   1:L PR[91] 10mm/sec CNT100;
   1:  PR[GP1:91,1] = PR[GP1:90,1] + 67.778;
   1:  PR[GP1:91,2] = PR[GP1:90,2] + -19.376;
   1:L PR[91] 10mm/sec CNT100;
   1:  PR[GP1:91,1] = PR[GP1:90,1] + 70.791;
   1:  PR[GP1:91,2] = PR[GP1:90,2] + -14.501;
   1:L PR[91] 10mm/sec CNT100;
   1:  PR[GP1:91,1] = PR[GP1:90,1] + 71.584;
   1:  PR[GP1:91,2] = PR[GP1:90,2] + -10.994;
   1:L PR[91] 10mm/sec CNT100;
   1:  PR[GP1:91,1] = PR[GP1:90,1] + 73.496;
   1:  PR[GP1:91,2] = PR[GP1:90,2] + -5.450;
   1:L PR[91] 10mm/sec CNT100;
   1:  PR[GP1:91,1] = PR[GP1:90,1] + 74.129;
   1:  PR[GP1:91,2] = PR[GP1:90,2] + 0.245;
   1:L PR[91] 10mm/sec CNT100;
   1:  PR[GP1:91,1] = PR[GP1:90,1] + 73.337;
   1:  PR[GP1:91,2] = PR[GP1:90,2] + 3.752;
   1:L PR[91] 10mm/sec CNT100;
   1:  PR[GP1:91,1] = PR[GP1:90,1] + 72.689;
   1:  PR[GP1:91,2] = PR[GP1:90,2] + 9.581;
   1:L PR[91] 10mm/sec CNT100;
   1:  PR[GP1:91,1] = PR[GP1:90,1] + 70.809;
   1:  PR[GP1:91,2] = PR[GP1:90,2] + 15.031;
   1:L PR[91] 10mm/sec CNT100;
   1:  PR[GP1:91,1] = PR[GP1:90,1] + 67.761;
   1:  PR[GP1:91,2] = PR[GP1:90,2] + 19.962;
   1:L PR[91] 10mm/sec CNT100;
   1:  PR[GP1:91,1] = PR[GP1:90,1] + 65.538;
   1:  PR[GP1:91,2] = PR[GP1:90,2] + 22.788;
   1:L PR[91] 10mm/sec CNT100;
   1:  PR[GP1:91,1] = PR[GP1:90,1] + 61.480;
   1:  PR[GP1:91,2] = PR[GP1:90,2] + 26.931;
   1:L PR[91] 10mm/sec CNT100;
   1:  PR[GP1:91,1] = PR[GP1:90,1] + 56.613;
   1:  PR[GP1:91,2] = PR[GP1:90,2] + 30.080;
   1:L PR[91] 10mm/sec CNT100;
   1:  PR[GP1:91,1] = PR[GP1:90,1] + 53.392;
   1:  PR[GP1:91,2] = PR[GP1:90,2] + 31.677;
   1:L PR[91] 10mm/sec CNT100;
   1:  PR[GP1:91,1] = PR[GP1:90,1] + 47.950;
   1:  PR[GP1:91,2] = PR[GP1:90,2] + 33.680;
   1:L PR[91] 10mm/sec CNT100;
   1:  PR[GP1:91,1] = PR[GP1:90,1] + 42.203;
   1:  PR[GP1:91,2] = PR[GP1:90,2] + 34.439;
   1:L PR[91] 10mm/sec CNT100;
   1:  PR[GP1:91,1] = PR[GP1:90,1] + 38.606;
   1:  PR[GP1:91,2] = PR[GP1:90,2] + 34.497;
   1:L PR[91] 10mm/sec CNT100;
   1:  PR[GP1:91,1] = PR[GP1:90,1] + 32.831;
   1:  PR[GP1:91,2] = PR[GP1:90,2] + 33.975;
   1:L PR[91] 10mm/sec CNT100;
   1:  PR[GP1:91,1] = PR[GP1:90,1] + 27.313;
   1:  PR[GP1:91,2] = PR[GP1:90,2] + 32.198;
   1:L PR[91] 10mm/sec CNT100;
   1:  PR[GP1:91,1] = PR[GP1:90,1] + 24.043;
   1:  PR[GP1:91,2] = PR[GP1:90,2] + 30.704;
   1:L PR[91] 10mm/sec CNT100;
   1:  PR[GP1:91,1] = PR[GP1:90,1] + 19.047;
   1:  PR[GP1:91,2] = PR[GP1:90,2] + 27.757;
   1:L PR[91] 10mm/sec CNT100;
   1:  PR[GP1:91,1] = PR[GP1:90,1] + 14.824;
   1:  PR[GP1:91,2] = PR[GP1:90,2] + 23.787;
   1:L PR[91] 10mm/sec CNT100;
   1:  PR[GP1:91,1] = PR[GP1:90,1] + 12.513;
   1:  PR[GP1:91,2] = PR[GP1:90,2] + 21.033;
   1:L PR[91] 10mm/sec CNT100;
   1:  PR[GP1:91,1] = PR[GP1:90,1] + 9.263;
   1:  PR[GP1:91,2] = PR[GP1:90,2] + 16.229;
   1:L PR[91] 10mm/sec CNT100;
   1:  PR[GP1:91,1] = PR[GP1:90,1] + 7.149;
   1:  PR[GP1:91,2] = PR[GP1:90,2] + 10.833;
   1:L PR[91] 10mm/sec CNT100;
   1:  PR[GP1:91,1] = PR[GP1:90,1] + 6.245;
   1:  PR[GP1:91,2] = PR[GP1:90,2] + 7.355;
   1:L PR[91] 10mm/sec CNT100;
   1:  PR[GP1:91,1] = PR[GP1:90,1] + 5.362;
   1:  PR[GP1:91,2] = PR[GP1:90,2] + 1.589;
   1:L PR[91] 10mm/sec CNT100;
   1:  PR[GP1:91,1] = PR[GP1:90,1] + 5.334;
   1:  PR[GP1:91,2] = PR[GP1:90,2] + 0.841;
   1:L PR[91] 10mm/sec CNT100;
   1:  PR[GP1:91,1] = PR[GP1:90,1] + -5.749;
   1:  PR[GP1:91,2] = PR[GP1:90,2] + 0.842;
   1:L PR[91] 10mm/sec CNT100;
   1:  PR[GP1:91,1] = PR[GP1:90,1] + -6.245;
   1:  PR[GP1:91,2] = PR[GP1:90,2] + 2.791;
   1:L PR[91] 10mm/sec CNT100;
   1:  PR[GP1:91,1] = PR[GP1:90,1] + -6.800;
   1:  PR[GP1:91,2] = PR[GP1:90,2] + 5.072;
   1:L PR[91] 10mm/sec CNT100;
   1:  PR[GP1:91,1] = PR[GP1:90,1] + -7.686;
   1:  PR[GP1:91,2] = PR[GP1:90,2] + 10.862;
   1:L PR[91] 10mm/sec CNT100;
   1:  PR[GP1:91,1] = PR[GP1:90,1] + -9.778;
   1:  PR[GP1:91,2] = PR[GP1:90,2] + 16.200;
   1:L PR[91] 10mm/sec CNT100;
   1:  PR[GP1:91,1] = PR[GP1:90,1] + -12.088;
   1:  PR[GP1:91,2] = PR[GP1:90,2] + 18.953;
   1:L PR[91] 10mm/sec CNT100;
   1:  PR[GP1:91,1] = PR[GP1:90,1] + -15.374;
   1:  PR[GP1:91,2] = PR[GP1:90,2] + 23.809;
   1:L PR[91] 10mm/sec CNT100;
   1:  PR[GP1:91,1] = PR[GP1:90,1] + -19.550;
   1:  PR[GP1:91,2] = PR[GP1:90,2] + 27.735;
   1:L PR[91] 10mm/sec CNT100;
   1:  PR[GP1:91,1] = PR[GP1:90,1] + -22.820;
   1:  PR[GP1:91,2] = PR[GP1:90,2] + 29.228;
   1:L PR[91] 10mm/sec CNT100;
   1:  PR[GP1:91,1] = PR[GP1:90,1] + -27.870;
   1:  PR[GP1:91,2] = PR[GP1:90,2] + 32.208;
   1:L PR[91] 10mm/sec CNT100;
   1:  PR[GP1:91,1] = PR[GP1:90,1] + -33.326;
   1:  PR[GP1:91,2] = PR[GP1:90,2] + 33.965;
   1:L PR[91] 10mm/sec CNT100;
   1:  PR[GP1:91,1] = PR[GP1:90,1] + -36.922;
   1:  PR[GP1:91,2] = PR[GP1:90,2] + 33.908;
   1:L PR[91] 10mm/sec CNT100;
   1:  PR[GP1:91,1] = PR[GP1:90,1] + -42.761;
   1:  PR[GP1:91,2] = PR[GP1:90,2] + 34.435;
   1:L PR[91] 10mm/sec CNT100;
   1:  PR[GP1:91,1] = PR[GP1:90,1] + -48.444;
   1:  PR[GP1:91,2] = PR[GP1:90,2] + 33.685;
   1:L PR[91] 10mm/sec CNT100;
   1:  PR[GP1:91,1] = PR[GP1:90,1] + -51.664;
   1:  PR[GP1:91,2] = PR[GP1:90,2] + 32.088;
   1:L PR[91] 10mm/sec CNT100;
   1:  PR[GP1:91,1] = PR[GP1:90,1] + -57.167;
   1:  PR[GP1:91,2] = PR[GP1:90,2] + 30.062;
   1:L PR[91] 10mm/sec CNT100;
   1:  PR[GP1:91,1] = PR[GP1:90,1] + -61.979;
   1:  PR[GP1:91,2] = PR[GP1:90,2] + 26.949;
   1:L PR[91] 10mm/sec CNT100;
   1:  PR[GP1:91,1] = PR[GP1:90,1] + -64.201;
   1:  PR[GP1:91,2] = PR[GP1:90,2] + 24.123;
   1:L PR[91] 10mm/sec CNT100;
   1:  PR[GP1:91,1] = PR[GP1:90,1] + -68.304;
   1:  PR[GP1:91,2] = PR[GP1:90,2] + 19.934;
   1:L PR[91] 10mm/sec CNT100;
   1:  PR[GP1:91,1] = PR[GP1:90,1] + -71.318;
   1:  PR[GP1:91,2] = PR[GP1:90,2] + 15.059;
   1:L PR[91] 10mm/sec CNT100;
   1:  PR[GP1:91,1] = PR[GP1:90,1] + -72.110;
   1:  PR[GP1:91,2] = PR[GP1:90,2] + 11.552;
   1:L PR[91] 10mm/sec CNT100;
   1:  PR[GP1:91,1] = PR[GP1:90,1] + -74.022;
   1:  PR[GP1:91,2] = PR[GP1:90,2] + 6.008;
   1:L PR[91] 10mm/sec CNT100;
   1:  PR[GP1:91,1] = PR[GP1:90,1] + -74.656;
   1:  PR[GP1:91,2] = PR[GP1:90,2] + 0.313;
   1:L PR[91] 10mm/sec CNT100;
   1:  PR[GP1:91,1] = PR[GP1:90,1] + -73.863;
   1:  PR[GP1:91,2] = PR[GP1:90,2] + -3.194;
   1:L PR[91] 10mm/sec CNT100;
   1:  PR[GP1:91,1] = PR[GP1:90,1] + -73.215;
   1:  PR[GP1:91,2] = PR[GP1:90,2] + -9.023;
   1:L PR[91] 10mm/sec CNT100;
   1:  PR[GP1:91,1] = PR[GP1:90,1] + -71.335;
   1:  PR[GP1:91,2] = PR[GP1:90,2] + -14.473;
   1:L PR[91] 10mm/sec CNT100;
   1:  PR[GP1:91,1] = PR[GP1:90,1] + -68.287;
   1:  PR[GP1:91,2] = PR[GP1:90,2] + -19.404;
   1:L PR[91] 10mm/sec CNT100;
   1:  PR[GP1:91,1] = PR[GP1:90,1] + -66.065;
   1:  PR[GP1:91,2] = PR[GP1:90,2] + -22.230;
   1:L PR[91] 10mm/sec CNT100;
   1:  PR[GP1:91,1] = PR[GP1:90,1] + -62.007;
   1:  PR[GP1:91,2] = PR[GP1:90,2] + -26.373;
   1:L PR[91] 10mm/sec CNT100;
   1:  PR[GP1:91,1] = PR[GP1:90,1] + -57.140;
   1:  PR[GP1:91,2] = PR[GP1:90,2] + -29.522;
   1:L PR[91] 10mm/sec CNT100;
   1:  PR[GP1:91,1] = PR[GP1:90,1] + -53.918;
   1:  PR[GP1:91,2] = PR[GP1:90,2] + -31.119;
   1:L PR[91] 10mm/sec CNT100;
   1:  PR[GP1:91,1] = PR[GP1:90,1] + -48.476;
   1:  PR[GP1:91,2] = PR[GP1:90,2] + -33.122;
   1:L PR[91] 10mm/sec CNT100;
   1:  PR[GP1:91,1] = PR[GP1:90,1] + -42.729;
   1:  PR[GP1:91,2] = PR[GP1:90,2] + -33.881;
   1:L PR[91] 10mm/sec CNT100;
   1:  PR[GP1:91,1] = PR[GP1:90,1] + -39.133;
   1:  PR[GP1:91,2] = PR[GP1:90,2] + -33.939;
   1:L PR[91] 10mm/sec CNT100;
   1:  PR[GP1:91,1] = PR[GP1:90,1] + -33.357;
   1:  PR[GP1:91,2] = PR[GP1:90,2] + -33.417;
   1:L PR[91] 10mm/sec CNT100;
   1:  PR[GP1:91,1] = PR[GP1:90,1] + -27.840;
   1:  PR[GP1:91,2] = PR[GP1:90,2] + -31.640;
   1:L PR[91] 10mm/sec CNT100;
   1:  PR[GP1:91,1] = PR[GP1:90,1] + -24.569;
   1:  PR[GP1:91,2] = PR[GP1:90,2] + -30.146;
   1:L PR[91] 10mm/sec CNT100;
   1:  PR[GP1:91,1] = PR[GP1:90,1] + -19.574;
   1:  PR[GP1:91,2] = PR[GP1:90,2] + -27.199;
   1:L PR[91] 10mm/sec CNT100;
   1:  PR[GP1:91,1] = PR[GP1:90,1] + -15.351;
   1:  PR[GP1:91,2] = PR[GP1:90,2] + -23.229;
   1:L PR[91] 10mm/sec CNT100;
   1:  PR[GP1:91,1] = PR[GP1:90,1] + -13.039;
   1:  PR[GP1:91,2] = PR[GP1:90,2] + -20.475;
   1:L PR[91] 10mm/sec CNT100;
   1:  PR[GP1:91,1] = PR[GP1:90,1] + -9.789;
   1:  PR[GP1:91,2] = PR[GP1:90,2] + -15.671;
   1:L PR[91] 10mm/sec CNT100;
   1:  PR[GP1:91,1] = PR[GP1:90,1] + -7.675;
   1:  PR[GP1:91,2] = PR[GP1:90,2] + -10.275;
   1:L PR[91] 10mm/sec CNT100;
   1:  PR[GP1:91,1] = PR[GP1:90,1] + -6.771;
   1:  PR[GP1:91,2] = PR[GP1:90,2] + -6.797;
   1:L PR[91] 10mm/sec CNT100;
   1:  PR[GP1:91,1] = PR[GP1:90,1] + -5.888;
   1:  PR[GP1:91,2] = PR[GP1:90,2] + -1.031;
   1:L PR[91] 10mm/sec CNT100;
   1:  PR[GP1:91,1] = PR[GP1:90,1] + -5.861;
   1:  PR[GP1:91,2] = PR[GP1:90,2] + -0.283;
   1:L PR[91] 10mm/sec CNT100;
   1:  PR[GP1:91,1] = PR[GP1:90,1] + 5.223;
   1:  PR[GP1:91,2] = PR[GP1:90,2] + -0.284;
   1:L PR[91] 10mm/sec CNT100;
   1:  PR[GP1:91,1] = PR[GP1:90,1] + 5.979;
   1:  PR[GP1:91,2] = PR[GP1:90,2] + -3.401;
   1:  PR[GP1:91,3] = PR[GP1:90,3] + 7.015;
   1:L PR[91] 10mm/sec CNT100;
   1:  PR[GP1:91,1] = PR[GP1:90,1] + 6.955;
   1:  PR[GP1:91,2] = PR[GP1:90,2] + -9.774;
   1:L PR[91] 10mm/sec CNT100;
   1:  PR[GP1:91,1] = PR[GP1:90,1] + 9.261;
   1:  PR[GP1:91,2] = PR[GP1:90,2] + -15.661;
   1:L PR[91] 10mm/sec CNT100;
   1:  PR[GP1:91,1] = PR[GP1:90,1] + 10.816;
   1:  PR[GP1:91,2] = PR[GP1:90,2] + -17.514;
   1:L PR[91] 10mm/sec CNT100;
   1:  PR[GP1:91,1] = PR[GP1:90,1] + 14.432;
   1:  PR[GP1:91,2] = PR[GP1:90,2] + -22.857;
   1:L PR[91] 10mm/sec CNT100;
   1:  PR[GP1:91,1] = PR[GP1:90,1] + 19.038;
   1:  PR[GP1:91,2] = PR[GP1:90,2] + -27.188;
   1:L PR[91] 10mm/sec CNT100;
   1:  PR[GP1:91,1] = PR[GP1:90,1] + 21.239;
   1:  PR[GP1:91,2] = PR[GP1:90,2] + -28.193;
   1:L PR[91] 10mm/sec CNT100;
   1:  PR[GP1:91,1] = PR[GP1:90,1] + 26.796;
   1:  PR[GP1:91,2] = PR[GP1:90,2] + -31.472;
   1:L PR[91] 10mm/sec CNT100;
   1:  PR[GP1:91,1] = PR[GP1:90,1] + 32.814;
   1:  PR[GP1:91,2] = PR[GP1:90,2] + -33.410;
   1:L PR[91] 10mm/sec CNT100;
   1:  PR[GP1:91,1] = PR[GP1:90,1] + 35.234;
   1:  PR[GP1:91,2] = PR[GP1:90,2] + -33.371;
   1:L PR[91] 10mm/sec CNT100;
   1:  PR[GP1:91,1] = PR[GP1:90,1] + 41.660;
   1:  PR[GP1:91,2] = PR[GP1:90,2] + -33.952;
   1:L PR[91] 10mm/sec CNT100;
   1:  PR[GP1:91,1] = PR[GP1:90,1] + 47.927;
   1:  PR[GP1:91,2] = PR[GP1:90,2] + -33.124;
   1:L PR[91] 10mm/sec CNT100;
   1:  PR[GP1:91,1] = PR[GP1:90,1] + 50.095;
   1:  PR[GP1:91,2] = PR[GP1:90,2] + -32.050;
   1:L PR[91] 10mm/sec CNT100;
   1:  PR[GP1:91,1] = PR[GP1:90,1] + 56.151;
   1:  PR[GP1:91,2] = PR[GP1:90,2] + -29.820;
   1:L PR[91] 10mm/sec CNT100;
   1:  PR[GP1:91,1] = PR[GP1:90,1] + 61.458;
   1:  PR[GP1:91,2] = PR[GP1:90,2] + -26.386;
   1:L PR[91] 10mm/sec CNT100;
   1:  PR[GP1:91,1] = PR[GP1:90,1] + 62.953;
   1:  PR[GP1:91,2] = PR[GP1:90,2] + -24.485;
   1:L PR[91] 10mm/sec CNT100;
   1:  PR[GP1:91,1] = PR[GP1:90,1] + 67.470;
   1:  PR[GP1:91,2] = PR[GP1:90,2] + -19.875;
   1:L PR[91] 10mm/sec CNT100;
   1:  PR[GP1:91,1] = PR[GP1:90,1] + 70.793;
   1:  PR[GP1:91,2] = PR[GP1:90,2] + -14.498;
   1:L PR[91] 10mm/sec CNT100;
   1:  PR[GP1:91,1] = PR[GP1:90,1] + 71.326;
   1:  PR[GP1:91,2] = PR[GP1:90,2] + -12.138;
   1:L PR[91] 10mm/sec CNT100;
   1:  PR[GP1:91,1] = PR[GP1:90,1] + 73.431;
   1:  PR[GP1:91,2] = PR[GP1:90,2] + -6.036;
   1:L PR[91] 10mm/sec CNT100;
   1:  PR[GP1:91,1] = PR[GP1:90,1] + 74.129;
   1:  PR[GP1:91,2] = PR[GP1:90,2] + 0.245;
   1:L PR[91] 10mm/sec CNT100;
   1:  PR[GP1:91,1] = PR[GP1:90,1] + 73.596;
   1:  PR[GP1:91,2] = PR[GP1:90,2] + 2.605;
   1:L PR[91] 10mm/sec CNT100;
   1:  PR[GP1:91,1] = PR[GP1:90,1] + 72.883;
   1:  PR[GP1:91,2] = PR[GP1:90,2] + 9.020;
   1:L PR[91] 10mm/sec CNT100;
   1:  PR[GP1:91,1] = PR[GP1:90,1] + 70.811;
   1:  PR[GP1:91,2] = PR[GP1:90,2] + 15.027;
   1:L PR[91] 10mm/sec CNT100;
   1:  PR[GP1:91,1] = PR[GP1:90,1] + 67.452;
   1:  PR[GP1:91,2] = PR[GP1:90,2] + 20.461;
   1:L PR[91] 10mm/sec CNT100;
   1:  PR[GP1:91,1] = PR[GP1:90,1] + 65.957;
   1:  PR[GP1:91,2] = PR[GP1:90,2] + 22.363;
   1:L PR[91] 10mm/sec CNT100;
   1:  PR[GP1:91,1] = PR[GP1:90,1] + 61.486;
   1:  PR[GP1:91,2] = PR[GP1:90,2] + 26.926;
   1:L PR[91] 10mm/sec CNT100;
   1:  PR[GP1:91,1] = PR[GP1:90,1] + 56.124;
   1:  PR[GP1:91,2] = PR[GP1:90,2] + 30.395;
   1:L PR[91] 10mm/sec CNT100;
   1:  PR[GP1:91,1] = PR[GP1:90,1] + 53.955;
   1:  PR[GP1:91,2] = PR[GP1:90,2] + 31.470;
   1:L PR[91] 10mm/sec CNT100;
   1:  PR[GP1:91,1] = PR[GP1:90,1] + 47.960;
   1:  PR[GP1:91,2] = PR[GP1:90,2] + 33.678;
   1:L PR[91] 10mm/sec CNT100;
   1:  PR[GP1:91,1] = PR[GP1:90,1] + 41.629;
   1:  PR[GP1:91,2] = PR[GP1:90,2] + 34.514;
   1:L PR[91] 10mm/sec CNT100;
   1:  PR[GP1:91,1] = PR[GP1:90,1] + 39.208;
   1:  PR[GP1:91,2] = PR[GP1:90,2] + 34.553;
   1:L PR[91] 10mm/sec CNT100;
   1:  PR[GP1:91,1] = PR[GP1:90,1] + 32.845;
   1:  PR[GP1:91,2] = PR[GP1:90,2] + 33.978;
   1:L PR[91] 10mm/sec CNT100;
   1:  PR[GP1:91,1] = PR[GP1:90,1] + 26.766;
   1:  PR[GP1:91,2] = PR[GP1:90,2] + 32.020;
   1:L PR[91] 10mm/sec CNT100;
   1:  PR[GP1:91,1] = PR[GP1:90,1] + 24.565;
   1:  PR[GP1:91,2] = PR[GP1:90,2] + 31.015;
   1:L PR[91] 10mm/sec CNT100;
   1:  PR[GP1:91,1] = PR[GP1:90,1] + 19.062;
   1:  PR[GP1:91,2] = PR[GP1:90,2] + 27.768;
   1:L PR[91] 10mm/sec CNT100;
   1:  PR[GP1:91,1] = PR[GP1:90,1] + 14.409;
   1:  PR[GP1:91,2] = PR[GP1:90,2] + 23.394;
   1:L PR[91] 10mm/sec CNT100;
   1:  PR[GP1:91,1] = PR[GP1:90,1] + 12.853;
   1:  PR[GP1:91,2] = PR[GP1:90,2] + 21.541;
   1:L PR[91] 10mm/sec CNT100;
   1:  PR[GP1:91,1] = PR[GP1:90,1] + 9.273;
   1:  PR[GP1:91,2] = PR[GP1:90,2] + 16.248;
   1:L PR[91] 10mm/sec CNT100;
   1:  PR[GP1:91,1] = PR[GP1:90,1] + 6.943;
   1:  PR[GP1:91,2] = PR[GP1:90,2] + 10.303;
   1:L PR[91] 10mm/sec CNT100;
   1:  PR[GP1:91,1] = PR[GP1:90,1] + 6.335;
   1:  PR[GP1:91,2] = PR[GP1:90,2] + 7.962;
   1:L PR[91] 10mm/sec CNT100;
   1:  PR[GP1:91,1] = PR[GP1:90,1] + 5.363;
   1:  PR[GP1:91,2] = PR[GP1:90,2] + 1.613;
   1:L PR[91] 10mm/sec CNT100;
   1:  PR[GP1:91,1] = PR[GP1:90,1] + 5.335;
   1:  PR[GP1:91,2] = PR[GP1:90,2] + 0.879;
   1:L PR[91] 10mm/sec CNT100;
   1:  PR[GP1:91,1] = PR[GP1:90,1] + -5.755;
   1:  PR[GP1:91,2] = PR[GP1:90,2] + 0.880;
   1:L PR[91] 10mm/sec CNT100;
   1:  PR[GP1:91,1] = PR[GP1:90,1] + -6.505;
   1:  PR[GP1:91,2] = PR[GP1:90,2] + 3.959;
   1:L PR[91] 10mm/sec CNT100;
   1:  PR[GP1:91,1] = PR[GP1:90,1] + -7.481;
   1:  PR[GP1:91,2] = PR[GP1:90,2] + 10.332;
   1:L PR[91] 10mm/sec CNT100;
   1:  PR[GP1:91,1] = PR[GP1:90,1] + -9.787;
   1:  PR[GP1:91,2] = PR[GP1:90,2] + 16.219;
   1:L PR[91] 10mm/sec CNT100;
   1:  PR[GP1:91,1] = PR[GP1:90,1] + -11.342;
   1:  PR[GP1:91,2] = PR[GP1:90,2] + 18.072;
   1:L PR[91] 10mm/sec CNT100;
   1:  PR[GP1:91,1] = PR[GP1:90,1] + -14.958;
   1:  PR[GP1:91,2] = PR[GP1:90,2] + 23.415;
   1:L PR[91] 10mm/sec CNT100;
   1:  PR[GP1:91,1] = PR[GP1:90,1] + -19.565;
   1:  PR[GP1:91,2] = PR[GP1:90,2] + 27.746;
   1:L PR[91] 10mm/sec CNT100;
   1:  PR[GP1:91,1] = PR[GP1:90,1] + -21.765;
   1:  PR[GP1:91,2] = PR[GP1:90,2] + 28.751;
   1:L PR[91] 10mm/sec CNT100;
   1:  PR[GP1:91,1] = PR[GP1:90,1] + -27.323;
   1:  PR[GP1:91,2] = PR[GP1:90,2] + 32.030;
   1:L PR[91] 10mm/sec CNT100;
   1:  PR[GP1:91,1] = PR[GP1:90,1] + -33.340;
   1:  PR[GP1:91,2] = PR[GP1:90,2] + 33.968;
   1:L PR[91] 10mm/sec CNT100;
   1:  PR[GP1:91,1] = PR[GP1:90,1] + -35.760;
   1:  PR[GP1:91,2] = PR[GP1:90,2] + 33.929;
   1:L PR[91] 10mm/sec CNT100;
   1:  PR[GP1:91,1] = PR[GP1:90,1] + -42.187;
   1:  PR[GP1:91,2] = PR[GP1:90,2] + 34.510;
   1:L PR[91] 10mm/sec CNT100;
   1:  PR[GP1:91,1] = PR[GP1:90,1] + -48.454;
   1:  PR[GP1:91,2] = PR[GP1:90,2] + 33.682;
   1:L PR[91] 10mm/sec CNT100;
   1:  PR[GP1:91,1] = PR[GP1:90,1] + -50.621;
   1:  PR[GP1:91,2] = PR[GP1:90,2] + 32.608;
   1:L PR[91] 10mm/sec CNT100;
   1:  PR[GP1:91,1] = PR[GP1:90,1] + -56.677;
   1:  PR[GP1:91,2] = PR[GP1:90,2] + 30.378;
   1:L PR[91] 10mm/sec CNT100;
   1:  PR[GP1:91,1] = PR[GP1:90,1] + -61.984;
   1:  PR[GP1:91,2] = PR[GP1:90,2] + 26.944;
   1:L PR[91] 10mm/sec CNT100;
   1:  PR[GP1:91,1] = PR[GP1:90,1] + -63.480;
   1:  PR[GP1:91,2] = PR[GP1:90,2] + 25.043;
   1:L PR[91] 10mm/sec CNT100;
   1:  PR[GP1:91,1] = PR[GP1:90,1] + -67.996;
   1:  PR[GP1:91,2] = PR[GP1:90,2] + 20.433;
   1:L PR[91] 10mm/sec CNT100;
   1:  PR[GP1:91,1] = PR[GP1:90,1] + -71.319;
   1:  PR[GP1:91,2] = PR[GP1:90,2] + 15.056;
   1:L PR[91] 10mm/sec CNT100;
   1:  PR[GP1:91,1] = PR[GP1:90,1] + -71.853;
   1:  PR[GP1:91,2] = PR[GP1:90,2] + 12.696;
   1:L PR[91] 10mm/sec CNT100;
   1:  PR[GP1:91,1] = PR[GP1:90,1] + -73.957;
   1:  PR[GP1:91,2] = PR[GP1:90,2] + 6.595;
   1:L PR[91] 10mm/sec CNT100;
   1:  PR[GP1:91,1] = PR[GP1:90,1] + -74.656;
   1:  PR[GP1:91,2] = PR[GP1:90,2] + 0.313;
   1:L PR[91] 10mm/sec CNT100;
   1:  PR[GP1:91,1] = PR[GP1:90,1] + -74.122;
   1:  PR[GP1:91,2] = PR[GP1:90,2] + -2.047;
   1:L PR[91] 10mm/sec CNT100;
   1:  PR[GP1:91,1] = PR[GP1:90,1] + -73.409;
   1:  PR[GP1:91,2] = PR[GP1:90,2] + -8.462;
   1:L PR[91] 10mm/sec CNT100;
   1:  PR[GP1:91,1] = PR[GP1:90,1] + -71.337;
   1:  PR[GP1:91,2] = PR[GP1:90,2] + -14.469;
   1:L PR[91] 10mm/sec CNT100;
   1:  PR[GP1:91,1] = PR[GP1:90,1] + -67.979;
   1:  PR[GP1:91,2] = PR[GP1:90,2] + -19.903;
   1:L PR[91] 10mm/sec CNT100;
   1:  PR[GP1:91,1] = PR[GP1:90,1] + -66.483;
   1:  PR[GP1:91,2] = PR[GP1:90,2] + -21.805;
   1:L PR[91] 10mm/sec CNT100;
   1:  PR[GP1:91,1] = PR[GP1:90,1] + -62.012;
   1:  PR[GP1:91,2] = PR[GP1:90,2] + -26.368;
   1:L PR[91] 10mm/sec CNT100;
   1:  PR[GP1:91,1] = PR[GP1:90,1] + -56.650;
   1:  PR[GP1:91,2] = PR[GP1:90,2] + -29.837;
   1:L PR[91] 10mm/sec CNT100;
   1:  PR[GP1:91,1] = PR[GP1:90,1] + -54.482;
   1:  PR[GP1:91,2] = PR[GP1:90,2] + -30.912;
   1:L PR[91] 10mm/sec CNT100;
   1:  PR[GP1:91,1] = PR[GP1:90,1] + -48.486;
   1:  PR[GP1:91,2] = PR[GP1:90,2] + -33.120;
   1:L PR[91] 10mm/sec CNT100;
   1:  PR[GP1:91,1] = PR[GP1:90,1] + -42.155;
   1:  PR[GP1:91,2] = PR[GP1:90,2] + -33.956;
   1:L PR[91] 10mm/sec CNT100;
   1:  PR[GP1:91,1] = PR[GP1:90,1] + -39.734;
   1:  PR[GP1:91,2] = PR[GP1:90,2] + -33.995;
   1:L PR[91] 10mm/sec CNT100;
   1:  PR[GP1:91,1] = PR[GP1:90,1] + -33.371;
   1:  PR[GP1:91,2] = PR[GP1:90,2] + -33.420;
   1:L PR[91] 10mm/sec CNT100;
   1:  PR[GP1:91,1] = PR[GP1:90,1] + -27.292;
   1:  PR[GP1:91,2] = PR[GP1:90,2] + -31.462;
   1:L PR[91] 10mm/sec CNT100;
   1:  PR[GP1:91,1] = PR[GP1:90,1] + -25.091;
   1:  PR[GP1:91,2] = PR[GP1:90,2] + -30.457;
   1:L PR[91] 10mm/sec CNT100;
   1:  PR[GP1:91,1] = PR[GP1:90,1] + -19.588;
   1:  PR[GP1:91,2] = PR[GP1:90,2] + -27.210;
   1:L PR[91] 10mm/sec CNT100;
   1:  PR[GP1:91,1] = PR[GP1:90,1] + -14.935;
   1:  PR[GP1:91,2] = PR[GP1:90,2] + -22.836;
   1:L PR[91] 10mm/sec CNT100;
   1:  PR[GP1:91,1] = PR[GP1:90,1] + -13.380;
   1:  PR[GP1:91,2] = PR[GP1:90,2] + -20.983;
   1:L PR[91] 10mm/sec CNT100;
   1:  PR[GP1:91,1] = PR[GP1:90,1] + -9.799;
   1:  PR[GP1:91,2] = PR[GP1:90,2] + -15.690;
   1:L PR[91] 10mm/sec CNT100;
   1:  PR[GP1:91,1] = PR[GP1:90,1] + -7.470;
   1:  PR[GP1:91,2] = PR[GP1:90,2] + -9.745;
   1:L PR[91] 10mm/sec CNT100;
   1:  PR[GP1:91,1] = PR[GP1:90,1] + -6.861;
   1:  PR[GP1:91,2] = PR[GP1:90,2] + -7.404;
   1:L PR[91] 10mm/sec CNT100;
   1:  PR[GP1:91,1] = PR[GP1:90,1] + -5.889;
   1:  PR[GP1:91,2] = PR[GP1:90,2] + -1.055;
   1:L PR[91] 10mm/sec CNT100;
   1:  PR[GP1:91,1] = PR[GP1:90,1] + -5.861;
   1:  PR[GP1:91,2] = PR[GP1:90,2] + -0.321;
   1:L PR[91] 10mm/sec CNT100;
   1:  PR[GP1:91,1] = PR[GP1:90,1] + 5.229;
   1:  PR[GP1:91,2] = PR[GP1:90,2] + -0.322;
   1:L PR[91] 10mm/sec CNT100;
   1:  PR[GP1:91,1] = PR[GP1:90,1] + 5.684;
   1:  PR[GP1:91,2] = PR[GP1:90,2] + -2.287;
   1:  PR[GP1:91,3] = PR[GP1:90,3] + 7.625;
   1:L PR[91] 10mm/sec CNT100;
   1:  PR[GP1:91,1] = PR[GP1:90,1] + 6.749;
   1:  PR[GP1:91,2] = PR[GP1:90,2] + -9.243;
   1:L PR[91] 10mm/sec CNT100;
   1:  PR[GP1:91,1] = PR[GP1:90,1] + 9.271;
   1:  PR[GP1:91,2] = PR[GP1:90,2] + -15.680;
   1:L PR[91] 10mm/sec CNT100;
   1:  PR[GP1:91,1] = PR[GP1:90,1] + 10.070;
   1:  PR[GP1:91,2] = PR[GP1:90,2] + -16.632;
   1:L PR[91] 10mm/sec CNT100;
   1:  PR[GP1:91,1] = PR[GP1:90,1] + 14.016;
   1:  PR[GP1:91,2] = PR[GP1:90,2] + -22.464;
   1:L PR[91] 10mm/sec CNT100;
   1:  PR[GP1:91,1] = PR[GP1:90,1] + 19.053;
   1:  PR[GP1:91,2] = PR[GP1:90,2] + -27.199;
   1:L PR[91] 10mm/sec CNT100;
   1:  PR[GP1:91,1] = PR[GP1:90,1] + 20.184;
   1:  PR[GP1:91,2] = PR[GP1:90,2] + -27.715;
   1:L PR[91] 10mm/sec CNT100;
   1:  PR[GP1:91,1] = PR[GP1:90,1] + 26.249;
   1:  PR[GP1:91,2] = PR[GP1:90,2] + -31.294;
   1:L PR[91] 10mm/sec CNT100;
   1:  PR[GP1:91,1] = PR[GP1:90,1] + 32.828;
   1:  PR[GP1:91,2] = PR[GP1:90,2] + -33.413;
   1:L PR[91] 10mm/sec CNT100;
   1:  PR[GP1:91,1] = PR[GP1:90,1] + 34.072;
   1:  PR[GP1:91,2] = PR[GP1:90,2] + -33.393;
   1:L PR[91] 10mm/sec CNT100;
   1:  PR[GP1:91,1] = PR[GP1:90,1] + 41.086;
   1:  PR[GP1:91,2] = PR[GP1:90,2] + -34.027;
   1:L PR[91] 10mm/sec CNT100;
   1:  PR[GP1:91,1] = PR[GP1:90,1] + 47.938;
   1:  PR[GP1:91,2] = PR[GP1:90,2] + -33.122;
   1:L PR[91] 10mm/sec CNT100;
   1:  PR[GP1:91,1] = PR[GP1:90,1] + 49.052;
   1:  PR[GP1:91,2] = PR[GP1:90,2] + -32.569;
   1:L PR[91] 10mm/sec CNT100;
   1:  PR[GP1:91,1] = PR[GP1:90,1] + 55.661;
   1:  PR[GP1:91,2] = PR[GP1:90,2] + -30.136;
   1:L PR[91] 10mm/sec CNT100;
   1:  PR[GP1:91,1] = PR[GP1:90,1] + 61.464;
   1:  PR[GP1:91,2] = PR[GP1:90,2] + -26.382;
   1:L PR[91] 10mm/sec CNT100;
   1:  PR[GP1:91,1] = PR[GP1:90,1] + 62.232;
   1:  PR[GP1:91,2] = PR[GP1:90,2] + -25.404;
   1:L PR[91] 10mm/sec CNT100;
   1:  PR[GP1:91,1] = PR[GP1:90,1] + 67.161;
   1:  PR[GP1:91,2] = PR[GP1:90,2] + -20.373;
   1:L PR[91] 10mm/sec CNT100;
   1:  PR[GP1:91,1] = PR[GP1:90,1] + 70.795;
   1:  PR[GP1:91,2] = PR[GP1:90,2] + -14.495;
   1:L PR[91] 10mm/sec CNT100;
   1:  PR[GP1:91,1] = PR[GP1:90,1] + 71.069;
   1:  PR[GP1:91,2] = PR[GP1:90,2] + -13.282;
   1:L PR[91] 10mm/sec CNT100;
   1:  PR[GP1:91,1] = PR[GP1:90,1] + 73.366;
   1:  PR[GP1:91,2] = PR[GP1:90,2] + -6.623;
   1:L PR[91] 10mm/sec CNT100;
   1:  PR[GP1:91,1] = PR[GP1:90,1] + 74.129;
   1:  PR[GP1:91,2] = PR[GP1:90,2] + 0.245;
   1:L PR[91] 10mm/sec CNT100;
   1:  PR[GP1:91,1] = PR[GP1:90,1] + 73.855;
   1:  PR[GP1:91,2] = PR[GP1:90,2] + 1.458;
   1:L PR[91] 10mm/sec CNT100;
   1:  PR[GP1:91,1] = PR[GP1:90,1] + 73.077;
   1:  PR[GP1:91,2] = PR[GP1:90,2] + 8.459;
   1:L PR[91] 10mm/sec CNT100;
   1:  PR[GP1:91,1] = PR[GP1:90,1] + 70.812;
   1:  PR[GP1:91,2] = PR[GP1:90,2] + 15.024;
   1:L PR[91] 10mm/sec CNT100;
   1:  PR[GP1:91,1] = PR[GP1:90,1] + 67.144;
   1:  PR[GP1:91,2] = PR[GP1:90,2] + 20.959;
   1:L PR[91] 10mm/sec CNT100;
   1:  PR[GP1:91,1] = PR[GP1:90,1] + 66.375;
   1:  PR[GP1:91,2] = PR[GP1:90,2] + 21.937;
   1:L PR[91] 10mm/sec CNT100;
   1:  PR[GP1:91,1] = PR[GP1:90,1] + 61.492;
   1:  PR[GP1:91,2] = PR[GP1:90,2] + 26.922;
   1:L PR[91] 10mm/sec CNT100;
   1:  PR[GP1:91,1] = PR[GP1:90,1] + 55.634;
   1:  PR[GP1:91,2] = PR[GP1:90,2] + 30.711;
   1:L PR[91] 10mm/sec CNT100;
   1:  PR[GP1:91,1] = PR[GP1:90,1] + 54.519;
   1:  PR[GP1:91,2] = PR[GP1:90,2] + 31.264;
   1:L PR[91] 10mm/sec CNT100;
   1:  PR[GP1:91,1] = PR[GP1:90,1] + 47.970;
   1:  PR[GP1:91,2] = PR[GP1:90,2] + 33.675;
   1:L PR[91] 10mm/sec CNT100;
   1:  PR[GP1:91,1] = PR[GP1:90,1] + 41.054;
   1:  PR[GP1:91,2] = PR[GP1:90,2] + 34.589;
   1:L PR[91] 10mm/sec CNT100;
   1:  PR[GP1:91,1] = PR[GP1:90,1] + 39.810;
   1:  PR[GP1:91,2] = PR[GP1:90,2] + 34.609;
   1:L PR[91] 10mm/sec CNT100;
   1:  PR[GP1:91,1] = PR[GP1:90,1] + 32.859;
   1:  PR[GP1:91,2] = PR[GP1:90,2] + 33.981;
   1:L PR[91] 10mm/sec CNT100;
   1:  PR[GP1:91,1] = PR[GP1:90,1] + 26.219;
   1:  PR[GP1:91,2] = PR[GP1:90,2] + 31.842;
   1:L PR[91] 10mm/sec CNT100;
   1:  PR[GP1:91,1] = PR[GP1:90,1] + 25.087;
   1:  PR[GP1:91,2] = PR[GP1:90,2] + 31.325;
   1:L PR[91] 10mm/sec CNT100;
   1:  PR[GP1:91,1] = PR[GP1:90,1] + 19.076;
   1:  PR[GP1:91,2] = PR[GP1:90,2] + 27.779;
   1:L PR[91] 10mm/sec CNT100;
   1:  PR[GP1:91,1] = PR[GP1:90,1] + 13.993;
   1:  PR[GP1:91,2] = PR[GP1:90,2] + 23.001;
   1:L PR[91] 10mm/sec CNT100;
   1:  PR[GP1:91,1] = PR[GP1:90,1] + 13.194;
   1:  PR[GP1:91,2] = PR[GP1:90,2] + 22.048;
   1:L PR[91] 10mm/sec CNT100;
   1:  PR[GP1:91,1] = PR[GP1:90,1] + 9.282;
   1:  PR[GP1:91,2] = PR[GP1:90,2] + 16.267;
   1:L PR[91] 10mm/sec CNT100;
   1:  PR[GP1:91,1] = PR[GP1:90,1] + 6.738;
   1:  PR[GP1:91,2] = PR[GP1:90,2] + 9.773;
   1:L PR[91] 10mm/sec CNT100;
   1:  PR[GP1:91,1] = PR[GP1:90,1] + 6.425;
   1:  PR[GP1:91,2] = PR[GP1:90,2] + 8.569;
   1:L PR[91] 10mm/sec CNT100;
   1:  PR[GP1:91,1] = PR[GP1:90,1] + 5.364;
   1:  PR[GP1:91,2] = PR[GP1:90,2] + 1.637;
   1:L PR[91] 10mm/sec CNT100;
   1:  PR[GP1:91,1] = PR[GP1:90,1] + 5.339;
   1:  PR[GP1:91,2] = PR[GP1:90,2] + 0.992;
   1:L PR[91] 10mm/sec CNT100;
   1:  PR[GP1:91,1] = PR[GP1:90,1] + -5.760;
   1:  PR[GP1:91,2] = PR[GP1:90,2] + 0.991;
   1:L PR[91] 10mm/sec CNT100;
   1:  PR[GP1:91,1] = PR[GP1:90,1] + -6.210;
   1:  PR[GP1:91,2] = PR[GP1:90,2] + 2.846;
   1:L PR[91] 10mm/sec CNT100;
   1:  PR[GP1:91,1] = PR[GP1:90,1] + -7.276;
   1:  PR[GP1:91,2] = PR[GP1:90,2] + 9.801;
   1:L PR[91] 10mm/sec CNT100;
   1:  PR[GP1:91,1] = PR[GP1:90,1] + -9.797;
   1:  PR[GP1:91,2] = PR[GP1:90,2] + 16.238;
   1:L PR[91] 10mm/sec CNT100;
   1:  PR[GP1:91,1] = PR[GP1:90,1] + -10.596;
   1:  PR[GP1:91,2] = PR[GP1:90,2] + 17.190;
   1:L PR[91] 10mm/sec CNT100;
   1:  PR[GP1:91,1] = PR[GP1:90,1] + -14.543;
   1:  PR[GP1:91,2] = PR[GP1:90,2] + 23.022;
   1:L PR[91] 10mm/sec CNT100;
   1:  PR[GP1:91,1] = PR[GP1:90,1] + -19.579;
   1:  PR[GP1:91,2] = PR[GP1:90,2] + 27.757;
   1:L PR[91] 10mm/sec CNT100;
   1:  PR[GP1:91,1] = PR[GP1:90,1] + -20.710;
   1:  PR[GP1:91,2] = PR[GP1:90,2] + 28.273;
   1:L PR[91] 10mm/sec CNT100;
   1:  PR[GP1:91,1] = PR[GP1:90,1] + -26.775;
   1:  PR[GP1:91,2] = PR[GP1:90,2] + 31.852;
   1:L PR[91] 10mm/sec CNT100;
   1:  PR[GP1:91,1] = PR[GP1:90,1] + -33.354;
   1:  PR[GP1:91,2] = PR[GP1:90,2] + 33.971;
   1:L PR[91] 10mm/sec CNT100;
   1:  PR[GP1:91,1] = PR[GP1:90,1] + -34.598;
   1:  PR[GP1:91,2] = PR[GP1:90,2] + 33.951;
   1:L PR[91] 10mm/sec CNT100;
   1:  PR[GP1:91,1] = PR[GP1:90,1] + -41.612;
   1:  PR[GP1:91,2] = PR[GP1:90,2] + 34.585;
   1:L PR[91] 10mm/sec CNT100;
   1:  PR[GP1:91,1] = PR[GP1:90,1] + -48.464;
   1:  PR[GP1:91,2] = PR[GP1:90,2] + 33.680;
   1:L PR[91] 10mm/sec CNT100;
   1:  PR[GP1:91,1] = PR[GP1:90,1] + -49.578;
   1:  PR[GP1:91,2] = PR[GP1:90,2] + 33.127;
   1:L PR[91] 10mm/sec CNT100;
   1:  PR[GP1:91,1] = PR[GP1:90,1] + -56.188;
   1:  PR[GP1:91,2] = PR[GP1:90,2] + 30.694;
   1:L PR[91] 10mm/sec CNT100;
   1:  PR[GP1:91,1] = PR[GP1:90,1] + -61.990;
   1:  PR[GP1:91,2] = PR[GP1:90,2] + 26.940;
   1:L PR[91] 10mm/sec CNT100;
   1:  PR[GP1:91,1] = PR[GP1:90,1] + -62.758;
   1:  PR[GP1:91,2] = PR[GP1:90,2] + 25.963;
   1:L PR[91] 10mm/sec CNT100;
   1:  PR[GP1:91,1] = PR[GP1:90,1] + -67.687;
   1:  PR[GP1:91,2] = PR[GP1:90,2] + 20.931;
   1:L PR[91] 10mm/sec CNT100;
   1:  PR[GP1:91,1] = PR[GP1:90,1] + -71.321;
   1:  PR[GP1:91,2] = PR[GP1:90,2] + 15.053;
   1:L PR[91] 10mm/sec CNT100;
   1:  PR[GP1:91,1] = PR[GP1:90,1] + -71.595;
   1:  PR[GP1:91,2] = PR[GP1:90,2] + 13.840;
   1:L PR[91] 10mm/sec CNT100;
   1:  PR[GP1:91,1] = PR[GP1:90,1] + -73.892;
   1:  PR[GP1:91,2] = PR[GP1:90,2] + 7.181;
   1:L PR[91] 10mm/sec CNT100;
   1:  PR[GP1:91,1] = PR[GP1:90,1] + -74.656;
   1:  PR[GP1:91,2] = PR[GP1:90,2] + 0.313;
   1:L PR[91] 10mm/sec CNT100;
   1:  PR[GP1:91,1] = PR[GP1:90,1] + -74.382;
   1:  PR[GP1:91,2] = PR[GP1:90,2] + -0.900;
   1:L PR[91] 10mm/sec CNT100;
   1:  PR[GP1:91,1] = PR[GP1:90,1] + -73.603;
   1:  PR[GP1:91,2] = PR[GP1:90,2] + -7.901;
   1:L PR[91] 10mm/sec CNT100;
   1:  PR[GP1:91,1] = PR[GP1:90,1] + -71.339;
   1:  PR[GP1:91,2] = PR[GP1:90,2] + -14.466;
   1:L PR[91] 10mm/sec CNT100;
   1:  PR[GP1:91,1] = PR[GP1:90,1] + -67.670;
   1:  PR[GP1:91,2] = PR[GP1:90,2] + -20.401;
   1:L PR[91] 10mm/sec CNT100;
   1:  PR[GP1:91,1] = PR[GP1:90,1] + -66.901;
   1:  PR[GP1:91,2] = PR[GP1:90,2] + -21.379;
   1:L PR[91] 10mm/sec CNT100;
   1:  PR[GP1:91,1] = PR[GP1:90,1] + -62.018;
   1:  PR[GP1:91,2] = PR[GP1:90,2] + -26.364;
   1:L PR[91] 10mm/sec CNT100;
   1:  PR[GP1:91,1] = PR[GP1:90,1] + -56.160;
   1:  PR[GP1:91,2] = PR[GP1:90,2] + -30.153;
   1:L PR[91] 10mm/sec CNT100;
   1:  PR[GP1:91,1] = PR[GP1:90,1] + -55.046;
   1:  PR[GP1:91,2] = PR[GP1:90,2] + -30.706;
   1:L PR[91] 10mm/sec CNT100;
   1:  PR[GP1:91,1] = PR[GP1:90,1] + -48.497;
   1:  PR[GP1:91,2] = PR[GP1:90,2] + -33.117;
   1:L PR[91] 10mm/sec CNT100;
   1:  PR[GP1:91,1] = PR[GP1:90,1] + -41.580;
   1:  PR[GP1:91,2] = PR[GP1:90,2] + -34.031;
   1:L PR[91] 10mm/sec CNT100;
   1:  PR[GP1:91,1] = PR[GP1:90,1] + -40.336;
   1:  PR[GP1:91,2] = PR[GP1:90,2] + -34.051;
   1:L PR[91] 10mm/sec CNT100;
   1:  PR[GP1:91,1] = PR[GP1:90,1] + -33.385;
   1:  PR[GP1:91,2] = PR[GP1:90,2] + -33.423;
   1:L PR[91] 10mm/sec CNT100;
   1:  PR[GP1:91,1] = PR[GP1:90,1] + -26.745;
   1:  PR[GP1:91,2] = PR[GP1:90,2] + -31.284;
   1:L PR[91] 10mm/sec CNT100;
   1:  PR[GP1:91,1] = PR[GP1:90,1] + -25.613;
   1:  PR[GP1:91,2] = PR[GP1:90,2] + -30.767;
   1:L PR[91] 10mm/sec CNT100;
   1:  PR[GP1:91,1] = PR[GP1:90,1] + -19.602;
   1:  PR[GP1:91,2] = PR[GP1:90,2] + -27.221;
   1:L PR[91] 10mm/sec CNT100;
   1:  PR[GP1:91,1] = PR[GP1:90,1] + -14.520;
   1:  PR[GP1:91,2] = PR[GP1:90,2] + -22.443;
   1:L PR[91] 10mm/sec CNT100;
   1:  PR[GP1:91,1] = PR[GP1:90,1] + -13.720;
   1:  PR[GP1:91,2] = PR[GP1:90,2] + -21.490;
   1:L PR[91] 10mm/sec CNT100;
   1:  PR[GP1:91,1] = PR[GP1:90,1] + -9.809;
   1:  PR[GP1:91,2] = PR[GP1:90,2] + -15.709;
   1:L PR[91] 10mm/sec CNT100;
   1:  PR[GP1:91,1] = PR[GP1:90,1] + -7.264;
   1:  PR[GP1:91,2] = PR[GP1:90,2] + -9.214;
   1:L PR[91] 10mm/sec CNT100;
   1:  PR[GP1:91,1] = PR[GP1:90,1] + -6.952;
   1:  PR[GP1:91,2] = PR[GP1:90,2] + -8.011;
   1:L PR[91] 10mm/sec CNT100;
   1:  PR[GP1:91,1] = PR[GP1:90,1] + -5.890;
   1:  PR[GP1:91,2] = PR[GP1:90,2] + -1.079;
   1:L PR[91] 10mm/sec CNT100;
   1:  PR[GP1:91,1] = PR[GP1:90,1] + -5.866;
   1:  PR[GP1:91,2] = PR[GP1:90,2] + -0.434;
   1:L PR[91] 10mm/sec CNT100;
   1:  PR[GP1:91,1] = PR[GP1:90,1] + 5.233;
   1:  PR[GP1:91,2] = PR[GP1:90,2] + -0.432;
   1:L PR[91] 10mm/sec CNT100;
   1:  PR[GP1:91,1] = PR[GP1:90,1] + 5.390;
   1:  PR[GP1:91,2] = PR[GP1:90,2] + -1.174;
   1:  PR[GP1:91,3] = PR[GP1:90,3] + 8.235;
   1:L PR[91] 10mm/sec CNT100;
   1:  PR[GP1:91,1] = PR[GP1:90,1] + 6.544;
   1:  PR[GP1:91,2] = PR[GP1:90,2] + -8.713;
   1:L PR[91] 10mm/sec CNT100;
   1:  PR[GP1:91,1] = PR[GP1:90,1] + 9.281;
   1:  PR[GP1:91,2] = PR[GP1:90,2] + -15.698;
   1:L PR[91] 10mm/sec CNT100;
   1:  PR[GP1:91,1] = PR[GP1:90,1] + 9.324;
   1:  PR[GP1:91,2] = PR[GP1:90,2] + -15.750;
   1:L PR[91] 10mm/sec CNT100;
   1:  PR[GP1:91,1] = PR[GP1:90,1] + 13.601;
   1:  PR[GP1:91,2] = PR[GP1:90,2] + -22.071;
   1:L PR[91] 10mm/sec CNT100;
   1:  PR[GP1:91,1] = PR[GP1:90,1] + 19.067;
   1:  PR[GP1:91,2] = PR[GP1:90,2] + -27.209;
   1:L PR[91] 10mm/sec CNT100;
   1:  PR[GP1:91,1] = PR[GP1:90,1] + 19.128;
   1:  PR[GP1:91,2] = PR[GP1:90,2] + -27.238;
   1:L PR[91] 10mm/sec CNT100;
   1:  PR[GP1:91,1] = PR[GP1:90,1] + 25.702;
   1:  PR[GP1:91,2] = PR[GP1:90,2] + -31.116;
   1:L PR[91] 10mm/sec CNT100;
   1:  PR[GP1:91,1] = PR[GP1:90,1] + 32.842;
   1:  PR[GP1:91,2] = PR[GP1:90,2] + -33.416;
   1:L PR[91] 10mm/sec CNT100;
   1:  PR[GP1:91,1] = PR[GP1:90,1] + 32.910;
   1:  PR[GP1:91,2] = PR[GP1:90,2] + -33.414;
   1:L PR[91] 10mm/sec CNT100;
   1:  PR[GP1:91,1] = PR[GP1:90,1] + 40.511;
   1:  PR[GP1:91,2] = PR[GP1:90,2] + -34.101;
   1:L PR[91] 10mm/sec CNT100;
   1:  PR[GP1:91,1] = PR[GP1:90,1] + 47.948;
   1:  PR[GP1:91,2] = PR[GP1:90,2] + -33.119;
   1:L PR[91] 10mm/sec CNT100;
   1:  PR[GP1:91,1] = PR[GP1:90,1] + 48.009;
   1:  PR[GP1:91,2] = PR[GP1:90,2] + -33.089;
   1:L PR[91] 10mm/sec CNT100;
   1:  PR[GP1:91,1] = PR[GP1:90,1] + 55.172;
   1:  PR[GP1:91,2] = PR[GP1:90,2] + -30.452;
   1:L PR[91] 10mm/sec CNT100;
   1:  PR[GP1:91,1] = PR[GP1:90,1] + 61.469;
   1:  PR[GP1:91,2] = PR[GP1:90,2] + -26.377;
   1:L PR[91] 10mm/sec CNT100;
   1:  PR[GP1:91,1] = PR[GP1:90,1] + 61.511;
   1:  PR[GP1:91,2] = PR[GP1:90,2] + -26.324;
   1:L PR[91] 10mm/sec CNT100;
   1:  PR[GP1:91,1] = PR[GP1:90,1] + 66.853;
   1:  PR[GP1:91,2] = PR[GP1:90,2] + -20.871;
   1:L PR[91] 10mm/sec CNT100;
   1:  PR[GP1:91,1] = PR[GP1:90,1] + 70.796;
   1:  PR[GP1:91,2] = PR[GP1:90,2] + -14.491;
   1:L PR[91] 10mm/sec CNT100;
   1:  PR[GP1:91,1] = PR[GP1:90,1] + 70.811;
   1:  PR[GP1:91,2] = PR[GP1:90,2] + -14.425;
   1:L PR[91] 10mm/sec CNT100;
   1:  PR[GP1:91,1] = PR[GP1:90,1] + 73.301;
   1:  PR[GP1:91,2] = PR[GP1:90,2] + -7.209;
   1:L PR[91] 10mm/sec CNT100;
   1:  PR[GP1:91,1] = PR[GP1:90,1] + 74.129;
   1:  PR[GP1:91,2] = PR[GP1:90,2] + 0.245;
   1:L PR[91] 10mm/sec CNT100;
   1:  PR[GP1:91,1] = PR[GP1:90,1] + 74.114;
   1:  PR[GP1:91,2] = PR[GP1:90,2] + 0.311;
   1:L PR[91] 10mm/sec CNT100;
   1:  PR[GP1:91,1] = PR[GP1:90,1] + 73.271;
   1:  PR[GP1:91,2] = PR[GP1:90,2] + 7.899;
   1:L PR[91] 10mm/sec CNT100;
   1:  PR[GP1:91,1] = PR[GP1:90,1] + 70.814;
   1:  PR[GP1:91,2] = PR[GP1:90,2] + 15.021;
   1:L PR[91] 10mm/sec CNT100;
   1:  PR[GP1:91,1] = PR[GP1:90,1] + 66.835;
   1:  PR[GP1:91,2] = PR[GP1:90,2] + 21.457;
   1:L PR[91] 10mm/sec CNT100;
   1:  PR[GP1:91,1] = PR[GP1:90,1] + 66.793;
   1:  PR[GP1:91,2] = PR[GP1:90,2] + 21.511;
   1:L PR[91] 10mm/sec CNT100;
   1:  PR[GP1:91,1] = PR[GP1:90,1] + 61.497;
   1:  PR[GP1:91,2] = PR[GP1:90,2] + 26.917;
   1:L PR[91] 10mm/sec CNT100;
   1:  PR[GP1:91,1] = PR[GP1:90,1] + 55.144;
   1:  PR[GP1:91,2] = PR[GP1:90,2] + 31.027;
   1:L PR[91] 10mm/sec CNT100;
   1:  PR[GP1:91,1] = PR[GP1:90,1] + 55.083;
   1:  PR[GP1:91,2] = PR[GP1:90,2] + 31.058;
   1:L PR[91] 10mm/sec CNT100;
   1:  PR[GP1:91,1] = PR[GP1:90,1] + 47.981;
   1:  PR[GP1:91,2] = PR[GP1:90,2] + 33.673;
   1:L PR[91] 10mm/sec CNT100;
   1:  PR[GP1:91,1] = PR[GP1:90,1] + 40.480;
   1:  PR[GP1:91,2] = PR[GP1:90,2] + 34.664;
   1:L PR[91] 10mm/sec CNT100;
   1:  PR[GP1:91,1] = PR[GP1:90,1] + 40.411;
   1:  PR[GP1:91,2] = PR[GP1:90,2] + 34.665;
   1:L PR[91] 10mm/sec CNT100;
   1:  PR[GP1:91,1] = PR[GP1:90,1] + 32.873;
   1:  PR[GP1:91,2] = PR[GP1:90,2] + 33.984;
   1:L PR[91] 10mm/sec CNT100;
   1:  PR[GP1:91,1] = PR[GP1:90,1] + 25.672;
   1:  PR[GP1:91,2] = PR[GP1:90,2] + 31.664;
   1:L PR[91] 10mm/sec CNT100;
   1:  PR[GP1:91,1] = PR[GP1:90,1] + 25.609;
   1:  PR[GP1:91,2] = PR[GP1:90,2] + 31.636;
   1:L PR[91] 10mm/sec CNT100;
   1:  PR[GP1:91,1] = PR[GP1:90,1] + 19.090;
   1:  PR[GP1:91,2] = PR[GP1:90,2] + 27.789;
   1:L PR[91] 10mm/sec CNT100;
   1:  PR[GP1:91,1] = PR[GP1:90,1] + 13.578;
   1:  PR[GP1:91,2] = PR[GP1:90,2] + 22.608;
   1:L PR[91] 10mm/sec CNT100;
   1:  PR[GP1:91,1] = PR[GP1:90,1] + 13.534;
   1:  PR[GP1:91,2] = PR[GP1:90,2] + 22.555;
   1:L PR[91] 10mm/sec CNT100;
   1:  PR[GP1:91,1] = PR[GP1:90,1] + 9.292;
   1:  PR[GP1:91,2] = PR[GP1:90,2] + 16.286;
   1:L PR[91] 10mm/sec CNT100;
   1:  PR[GP1:91,1] = PR[GP1:90,1] + 6.533;
   1:  PR[GP1:91,2] = PR[GP1:90,2] + 9.242;
   1:L PR[91] 10mm/sec CNT100;
   1:  PR[GP1:91,1] = PR[GP1:90,1] + 6.515;
   1:  PR[GP1:91,2] = PR[GP1:90,2] + 9.176;
   1:L PR[91] 10mm/sec CNT100;
   1:  PR[GP1:91,1] = PR[GP1:90,1] + 5.281;
   1:  PR[GP1:91,2] = PR[GP1:90,2] + 1.108;
   1:L PR[91] 10mm/sec CNT100;
   1:  PR[GP1:91,1] = PR[GP1:90,1] + -5.764;
   1:  PR[GP1:91,2] = PR[GP1:90,2] + 1.107;
   1:L PR[91] 10mm/sec CNT100;
   1:  PR[GP1:91,1] = PR[GP1:90,1] + -5.916;
   1:  PR[GP1:91,2] = PR[GP1:90,2] + 1.732;
   1:L PR[91] 10mm/sec CNT100;
   1:  PR[GP1:91,1] = PR[GP1:90,1] + -7.070;
   1:  PR[GP1:91,2] = PR[GP1:90,2] + 9.271;
   1:L PR[91] 10mm/sec CNT100;
   1:  PR[GP1:91,1] = PR[GP1:90,1] + -9.807;
   1:  PR[GP1:91,2] = PR[GP1:90,2] + 16.257;
   1:L PR[91] 10mm/sec CNT100;
   1:  PR[GP1:91,1] = PR[GP1:90,1] + -9.850;
   1:  PR[GP1:91,2] = PR[GP1:90,2] + 16.308;
   1:L PR[91] 10mm/sec CNT100;
   1:  PR[GP1:91,1] = PR[GP1:90,1] + -14.127;
   1:  PR[GP1:91,2] = PR[GP1:90,2] + 22.629;
   1:L PR[91] 10mm/sec CNT100;
   1:  PR[GP1:91,1] = PR[GP1:90,1] + -19.593;
   1:  PR[GP1:91,2] = PR[GP1:90,2] + 27.767;
   1:L PR[91] 10mm/sec CNT100;
   1:  PR[GP1:91,1] = PR[GP1:90,1] + -19.655;
   1:  PR[GP1:91,2] = PR[GP1:90,2] + 27.796;
   1:L PR[91] 10mm/sec CNT100;
   1:  PR[GP1:91,1] = PR[GP1:90,1] + -26.228;
   1:  PR[GP1:91,2] = PR[GP1:90,2] + 31.674;
   1:L PR[91] 10mm/sec CNT100;
   1:  PR[GP1:91,1] = PR[GP1:90,1] + -33.369;
   1:  PR[GP1:91,2] = PR[GP1:90,2] + 33.974;
   1:L PR[91] 10mm/sec CNT100;
   1:  PR[GP1:91,1] = PR[GP1:90,1] + -33.436;
   1:  PR[GP1:91,2] = PR[GP1:90,2] + 33.972;
   1:L PR[91] 10mm/sec CNT100;
   1:  PR[GP1:91,1] = PR[GP1:90,1] + -41.038;
   1:  PR[GP1:91,2] = PR[GP1:90,2] + 34.659;
   1:L PR[91] 10mm/sec CNT100;
   1:  PR[GP1:91,1] = PR[GP1:90,1] + -48.474;
   1:  PR[GP1:91,2] = PR[GP1:90,2] + 33.677;
   1:L PR[91] 10mm/sec CNT100;
   1:  PR[GP1:91,1] = PR[GP1:90,1] + -48.535;
   1:  PR[GP1:91,2] = PR[GP1:90,2] + 33.647;
   1:L PR[91] 10mm/sec CNT100;
   1:  PR[GP1:91,1] = PR[GP1:90,1] + -55.698;
   1:  PR[GP1:91,2] = PR[GP1:90,2] + 31.010;
   1:L PR[91] 10mm/sec CNT100;
   1:  PR[GP1:91,1] = PR[GP1:90,1] + -61.996;
   1:  PR[GP1:91,2] = PR[GP1:90,2] + 26.935;
   1:L PR[91] 10mm/sec CNT100;
   1:  PR[GP1:91,1] = PR[GP1:90,1] + -62.037;
   1:  PR[GP1:91,2] = PR[GP1:90,2] + 26.882;
   1:L PR[91] 10mm/sec CNT100;
   1:  PR[GP1:91,1] = PR[GP1:90,1] + -67.379;
   1:  PR[GP1:91,2] = PR[GP1:90,2] + 21.429;
   1:L PR[91] 10mm/sec CNT100;
   1:  PR[GP1:91,1] = PR[GP1:90,1] + -71.323;
   1:  PR[GP1:91,2] = PR[GP1:90,2] + 15.049;
   1:L PR[91] 10mm/sec CNT100;
   1:  PR[GP1:91,1] = PR[GP1:90,1] + -71.337;
   1:  PR[GP1:91,2] = PR[GP1:90,2] + 14.983;
   1:L PR[91] 10mm/sec CNT100;
   1:  PR[GP1:91,1] = PR[GP1:90,1] + -73.827;
   1:  PR[GP1:91,2] = PR[GP1:90,2] + 7.767;
   1:L PR[91] 10mm/sec CNT100;
   1:  PR[GP1:91,1] = PR[GP1:90,1] + -74.656;
   1:  PR[GP1:91,2] = PR[GP1:90,2] + 0.313;
   1:L PR[91] 10mm/sec CNT100;
   1:  PR[GP1:91,1] = PR[GP1:90,1] + -74.641;
   1:  PR[GP1:91,2] = PR[GP1:90,2] + 0.247;
   1:L PR[91] 10mm/sec CNT100;
   1:  PR[GP1:91,1] = PR[GP1:90,1] + -73.797;
   1:  PR[GP1:91,2] = PR[GP1:90,2] + -7.341;
   1:L PR[91] 10mm/sec CNT100;
   1:  PR[GP1:91,1] = PR[GP1:90,1] + -71.340;
   1:  PR[GP1:91,2] = PR[GP1:90,2] + -14.463;
   1:L PR[91] 10mm/sec CNT100;
   1:  PR[GP1:91,1] = PR[GP1:90,1] + -67.362;
   1:  PR[GP1:91,2] = PR[GP1:90,2] + -20.899;
   1:L PR[91] 10mm/sec CNT100;
   1:  PR[GP1:91,1] = PR[GP1:90,1] + -67.319;
   1:  PR[GP1:91,2] = PR[GP1:90,2] + -20.953;
   1:L PR[91] 10mm/sec CNT100;
   1:  PR[GP1:91,1] = PR[GP1:90,1] + -62.023;
   1:  PR[GP1:91,2] = PR[GP1:90,2] + -26.359;
   1:L PR[91] 10mm/sec CNT100;
   1:  PR[GP1:91,1] = PR[GP1:90,1] + -55.671;
   1:  PR[GP1:91,2] = PR[GP1:90,2] + -30.469;
   1:L PR[91] 10mm/sec CNT100;
   1:  PR[GP1:91,1] = PR[GP1:90,1] + -55.609;
   1:  PR[GP1:91,2] = PR[GP1:90,2] + -30.500;
   1:L PR[91] 10mm/sec CNT100;
   1:  PR[GP1:91,1] = PR[GP1:90,1] + -48.507;
   1:  PR[GP1:91,2] = PR[GP1:90,2] + -33.115;
   1:L PR[91] 10mm/sec CNT100;
   1:  PR[GP1:91,1] = PR[GP1:90,1] + -41.006;
   1:  PR[GP1:91,2] = PR[GP1:90,2] + -34.106;
   1:L PR[91] 10mm/sec CNT100;
   1:  PR[GP1:91,1] = PR[GP1:90,1] + -40.938;
   1:  PR[GP1:91,2] = PR[GP1:90,2] + -34.107;
   1:L PR[91] 10mm/sec CNT100;
   1:  PR[GP1:91,1] = PR[GP1:90,1] + -33.399;
   1:  PR[GP1:91,2] = PR[GP1:90,2] + -33.425;
   1:L PR[91] 10mm/sec CNT100;
   1:  PR[GP1:91,1] = PR[GP1:90,1] + -26.198;
   1:  PR[GP1:91,2] = PR[GP1:90,2] + -31.106;
   1:L PR[91] 10mm/sec CNT100;
   1:  PR[GP1:91,1] = PR[GP1:90,1] + -26.136;
   1:  PR[GP1:91,2] = PR[GP1:90,2] + -31.078;
   1:L PR[91] 10mm/sec CNT100;
   1:  PR[GP1:91,1] = PR[GP1:90,1] + -19.617;
   1:  PR[GP1:91,2] = PR[GP1:90,2] + -27.231;
   1:L PR[91] 10mm/sec CNT100;
   1:  PR[GP1:91,1] = PR[GP1:90,1] + -14.104;
   1:  PR[GP1:91,2] = PR[GP1:90,2] + -22.050;
   1:L PR[91] 10mm/sec CNT100;
   1:  PR[GP1:91,1] = PR[GP1:90,1] + -14.060;
   1:  PR[GP1:91,2] = PR[GP1:90,2] + -21.997;
   1:L PR[91] 10mm/sec CNT100;
   1:  PR[GP1:91,1] = PR[GP1:90,1] + -9.818;
   1:  PR[GP1:91,2] = PR[GP1:90,2] + -15.728;
   1:L PR[91] 10mm/sec CNT100;
   1:  PR[GP1:91,1] = PR[GP1:90,1] + -7.059;
   1:  PR[GP1:91,2] = PR[GP1:90,2] + -8.684;
   1:L PR[91] 10mm/sec CNT100;
   1:  PR[GP1:91,1] = PR[GP1:90,1] + -7.042;
   1:  PR[GP1:91,2] = PR[GP1:90,2] + -8.618;
   1:L PR[91] 10mm/sec CNT100;
   1:  PR[GP1:91,1] = PR[GP1:90,1] + -5.808;
   1:  PR[GP1:91,2] = PR[GP1:90,2] + -0.550;
   1:L PR[91] 10mm/sec CNT100;
   1:  PR[GP1:91,1] = PR[GP1:90,1] + 5.238;
   1:  PR[GP1:91,2] = PR[GP1:90,2] + -0.549;
   1:L PR[91] 10mm/sec CNT100;
   1:  PR[GP1:91,1] = PR[GP1:90,1] + 5.987;
   1:  PR[GP1:91,2] = PR[GP1:90,2] + -5.336;
   1:  PR[GP1:91,3] = PR[GP1:90,3] + 8.845;
   1:L PR[91] 10mm/sec CNT100;
   1:  PR[GP1:91,1] = PR[GP1:90,1] + 6.415;
   1:  PR[GP1:91,2] = PR[GP1:90,2] + -8.334;
   1:L PR[91] 10mm/sec CNT100;
   1:  PR[GP1:91,1] = PR[GP1:90,1] + 9.000;
   1:  PR[GP1:91,2] = PR[GP1:90,2] + -14.933;
   1:L PR[91] 10mm/sec CNT100;
   1:  PR[GP1:91,1] = PR[GP1:90,1] + 9.300;
   1:  PR[GP1:91,2] = PR[GP1:90,2] + -15.812;
   1:L PR[91] 10mm/sec CNT100;
   1:  PR[GP1:91,1] = PR[GP1:90,1] + 13.253;
   1:  PR[GP1:91,2] = PR[GP1:90,2] + -21.655;
   1:L PR[91] 10mm/sec CNT100;
   1:  PR[GP1:91,1] = PR[GP1:90,1] + 13.810;
   1:  PR[GP1:91,2] = PR[GP1:90,2] + -22.316;
   1:L PR[91] 10mm/sec CNT100;
   1:  PR[GP1:91,1] = PR[GP1:90,1] + 18.987;
   1:  PR[GP1:91,2] = PR[GP1:90,2] + -27.183;
   1:L PR[91] 10mm/sec CNT100;
   1:  PR[GP1:91,1] = PR[GP1:90,1] + 25.127;
   1:  PR[GP1:91,2] = PR[GP1:90,2] + -30.805;
   1:L PR[91] 10mm/sec CNT100;
   1:  PR[GP1:91,1] = PR[GP1:90,1] + 25.835;
   1:  PR[GP1:91,2] = PR[GP1:90,2] + -31.187;
   1:L PR[91] 10mm/sec CNT100;
   1:  PR[GP1:91,1] = PR[GP1:90,1] + 32.625;
   1:  PR[GP1:91,2] = PR[GP1:90,2] + -33.374;
   1:L PR[91] 10mm/sec CNT100;
   1:  PR[GP1:91,1] = PR[GP1:90,1] + 39.792;
   1:  PR[GP1:91,2] = PR[GP1:90,2] + -34.022;
   1:L PR[91] 10mm/sec CNT100;
   1:  PR[GP1:91,1] = PR[GP1:90,1] + 40.525;
   1:  PR[GP1:91,2] = PR[GP1:90,2] + -34.109;
   1:L PR[91] 10mm/sec CNT100;
   1:  PR[GP1:91,1] = PR[GP1:90,1] + 47.650;
   1:  PR[GP1:91,2] = PR[GP1:90,2] + -33.168;
   1:L PR[91] 10mm/sec CNT100;
   1:  PR[GP1:91,1] = PR[GP1:90,1] + 48.270;
   1:  PR[GP1:91,2] = PR[GP1:90,2] + -33.007;
   1:L PR[91] 10mm/sec CNT100;
   1:  PR[GP1:91,1] = PR[GP1:90,1] + 55.063;
   1:  PR[GP1:91,2] = PR[GP1:90,2] + -30.506;
   1:L PR[91] 10mm/sec CNT100;
   1:  PR[GP1:91,1] = PR[GP1:90,1] + 61.151;
   1:  PR[GP1:91,2] = PR[GP1:90,2] + -26.567;
   1:L PR[91] 10mm/sec CNT100;
   1:  PR[GP1:91,1] = PR[GP1:90,1] + 61.633;
   1:  PR[GP1:91,2] = PR[GP1:90,2] + -26.216;
   1:L PR[91] 10mm/sec CNT100;
   1:  PR[GP1:91,1] = PR[GP1:90,1] + 66.703;
   1:  PR[GP1:91,2] = PR[GP1:90,2] + -21.041;
   1:L PR[91] 10mm/sec CNT100;
   1:  PR[GP1:91,1] = PR[GP1:90,1] + 70.839;
   1:  PR[GP1:91,2] = PR[GP1:90,2] + -14.362;
   1:L PR[91] 10mm/sec CNT100;
   1:  PR[GP1:91,1] = PR[GP1:90,1] + 73.201;
   1:  PR[GP1:91,2] = PR[GP1:90,2] + -7.516;
   1:L PR[91] 10mm/sec CNT100;
   1:  PR[GP1:91,1] = PR[GP1:90,1] + 74.011;
   1:  PR[GP1:91,2] = PR[GP1:90,2] + -0.229;
   1:L PR[91] 10mm/sec CNT100;
   1:  PR[GP1:91,1] = PR[GP1:90,1] + 74.112;
   1:  PR[GP1:91,2] = PR[GP1:90,2] + 0.302;
   1:L PR[91] 10mm/sec CNT100;
   1:  PR[GP1:91,1] = PR[GP1:90,1] + 73.308;
   1:  PR[GP1:91,2] = PR[GP1:90,2] + 7.534;
   1:L PR[91] 10mm/sec CNT100;
   1:  PR[GP1:91,1] = PR[GP1:90,1] + 73.209;
   1:  PR[GP1:91,2] = PR[GP1:90,2] + 8.052;
   1:L PR[91] 10mm/sec CNT100;
   1:  PR[GP1:91,1] = PR[GP1:90,1] + 70.839;
   1:  PR[GP1:91,2] = PR[GP1:90,2] + 14.920;
   1:L PR[91] 10mm/sec CNT100;
   1:  PR[GP1:91,1] = PR[GP1:90,1] + 66.998;
   1:  PR[GP1:91,2] = PR[GP1:90,2] + 21.135;
   1:L PR[91] 10mm/sec CNT100;
   1:  PR[GP1:91,1] = PR[GP1:90,1] + 66.705;
   1:  PR[GP1:91,2] = PR[GP1:90,2] + 21.597;
   1:L PR[91] 10mm/sec CNT100;
   1:  PR[GP1:91,1] = PR[GP1:90,1] + 61.645;
   1:  PR[GP1:91,2] = PR[GP1:90,2] + 26.762;
   1:L PR[91] 10mm/sec CNT100;
   1:  PR[GP1:91,1] = PR[GP1:90,1] + 55.507;
   1:  PR[GP1:91,2] = PR[GP1:90,2] + 30.734;
   1:L PR[91] 10mm/sec CNT100;
   1:  PR[GP1:91,1] = PR[GP1:90,1] + 55.047;
   1:  PR[GP1:91,2] = PR[GP1:90,2] + 31.070;
   1:L PR[91] 10mm/sec CNT100;
   1:  PR[GP1:91,1] = PR[GP1:90,1] + 48.270;
   1:  PR[GP1:91,2] = PR[GP1:90,2] + 33.565;
   1:L PR[91] 10mm/sec CNT100;
   1:  PR[GP1:91,1] = PR[GP1:90,1] + 47.650;
   1:  PR[GP1:91,2] = PR[GP1:90,2] + 33.726;
   1:L PR[91] 10mm/sec CNT100;
   1:  PR[GP1:91,1] = PR[GP1:90,1] + 40.517;
   1:  PR[GP1:91,2] = PR[GP1:90,2] + 34.668;
   1:L PR[91] 10mm/sec CNT100;
   1:  PR[GP1:91,1] = PR[GP1:90,1] + 33.323;
   1:  PR[GP1:91,2] = PR[GP1:90,2] + 34.018;
   1:L PR[91] 10mm/sec CNT100;
   1:  PR[GP1:91,1] = PR[GP1:90,1] + 32.633;
   1:  PR[GP1:91,2] = PR[GP1:90,2] + 33.935;
   1:L PR[91] 10mm/sec CNT100;
   1:  PR[GP1:91,1] = PR[GP1:90,1] + 25.846;
   1:  PR[GP1:91,2] = PR[GP1:90,2] + 31.749;
   1:L PR[91] 10mm/sec CNT100;
   1:  PR[GP1:91,1] = PR[GP1:90,1] + 19.645;
   1:  PR[GP1:91,2] = PR[GP1:90,2] + 28.090;
   1:L PR[91] 10mm/sec CNT100;
   1:  PR[GP1:91,1] = PR[GP1:90,1] + 18.978;
   1:  PR[GP1:91,2] = PR[GP1:90,2] + 27.732;
   1:L PR[91] 10mm/sec CNT100;
   1:  PR[GP1:91,1] = PR[GP1:90,1] + 13.810;
   1:  PR[GP1:91,2] = PR[GP1:90,2] + 22.874;
   1:L PR[91] 10mm/sec CNT100;
   1:  PR[GP1:91,1] = PR[GP1:90,1] + 13.253;
   1:  PR[GP1:91,2] = PR[GP1:90,2] + 22.213;
   1:L PR[91] 10mm/sec CNT100;
   1:  PR[GP1:91,1] = PR[GP1:90,1] + 9.292;
   1:  PR[GP1:91,2] = PR[GP1:90,2] + 16.359;
   1:L PR[91] 10mm/sec CNT100;
   1:  PR[GP1:91,1] = PR[GP1:90,1] + 6.707;
   1:  PR[GP1:91,2] = PR[GP1:90,2] + 9.762;
   1:L PR[91] 10mm/sec CNT100;
   1:  PR[GP1:91,1] = PR[GP1:90,1] + 6.416;
   1:  PR[GP1:91,2] = PR[GP1:90,2] + 8.903;
   1:L PR[91] 10mm/sec CNT100;
   1:  PR[GP1:91,1] = PR[GP1:90,1] + 5.359;
   1:  PR[GP1:91,2] = PR[GP1:90,2] + 2.000;
   1:L PR[91] 10mm/sec CNT100;
   1:  PR[GP1:91,1] = PR[GP1:90,1] + 5.504;
   1:  PR[GP1:91,2] = PR[GP1:90,2] + 1.295;
   1:L PR[91] 10mm/sec CNT100;
   1:  PR[GP1:91,1] = PR[GP1:90,1] + -5.809;
   1:  PR[GP1:91,2] = PR[GP1:90,2] + 1.296;
   1:L PR[91] 10mm/sec CNT100;
   1:  PR[GP1:91,1] = PR[GP1:90,1] + -6.513;
   1:  PR[GP1:91,2] = PR[GP1:90,2] + 5.891;
   1:L PR[91] 10mm/sec CNT100;
   1:  PR[GP1:91,1] = PR[GP1:90,1] + -6.941;
   1:  PR[GP1:91,2] = PR[GP1:90,2] + 8.892;
   1:L PR[91] 10mm/sec CNT100;
   1:  PR[GP1:91,1] = PR[GP1:90,1] + -9.526;
   1:  PR[GP1:91,2] = PR[GP1:90,2] + 15.491;
   1:L PR[91] 10mm/sec CNT100;
   1:  PR[GP1:91,1] = PR[GP1:90,1] + -9.826;
   1:  PR[GP1:91,2] = PR[GP1:90,2] + 16.371;
   1:L PR[91] 10mm/sec CNT100;
   1:  PR[GP1:91,1] = PR[GP1:90,1] + -13.779;
   1:  PR[GP1:91,2] = PR[GP1:90,2] + 22.213;
   1:L PR[91] 10mm/sec CNT100;
   1:  PR[GP1:91,1] = PR[GP1:90,1] + -14.336;
   1:  PR[GP1:91,2] = PR[GP1:90,2] + 22.874;
   1:L PR[91] 10mm/sec CNT100;
   1:  PR[GP1:91,1] = PR[GP1:90,1] + -19.514;
   1:  PR[GP1:91,2] = PR[GP1:90,2] + 27.741;
   1:L PR[91] 10mm/sec CNT100;
   1:  PR[GP1:91,1] = PR[GP1:90,1] + -25.654;
   1:  PR[GP1:91,2] = PR[GP1:90,2] + 31.364;
   1:L PR[91] 10mm/sec CNT100;
   1:  PR[GP1:91,1] = PR[GP1:90,1] + -26.362;
   1:  PR[GP1:91,2] = PR[GP1:90,2] + 31.745;
   1:L PR[91] 10mm/sec CNT100;
   1:  PR[GP1:91,1] = PR[GP1:90,1] + -33.151;
   1:  PR[GP1:91,2] = PR[GP1:90,2] + 33.932;
   1:L PR[91] 10mm/sec CNT100;
   1:  PR[GP1:91,1] = PR[GP1:90,1] + -40.319;
   1:  PR[GP1:91,2] = PR[GP1:90,2] + 34.580;
   1:L PR[91] 10mm/sec CNT100;
   1:  PR[GP1:91,1] = PR[GP1:90,1] + -41.052;
   1:  PR[GP1:91,2] = PR[GP1:90,2] + 34.667;
   1:L PR[91] 10mm/sec CNT100;
   1:  PR[GP1:91,1] = PR[GP1:90,1] + -48.177;
   1:  PR[GP1:91,2] = PR[GP1:90,2] + 33.726;
   1:L PR[91] 10mm/sec CNT100;
   1:  PR[GP1:91,1] = PR[GP1:90,1] + -48.797;
   1:  PR[GP1:91,2] = PR[GP1:90,2] + 33.565;
   1:L PR[91] 10mm/sec CNT100;
   1:  PR[GP1:91,1] = PR[GP1:90,1] + -55.589;
   1:  PR[GP1:91,2] = PR[GP1:90,2] + 31.064;
   1:L PR[91] 10mm/sec CNT100;
   1:  PR[GP1:91,1] = PR[GP1:90,1] + -61.678;
   1:  PR[GP1:91,2] = PR[GP1:90,2] + 27.125;
   1:L PR[91] 10mm/sec CNT100;
   1:  PR[GP1:91,1] = PR[GP1:90,1] + -62.160;
   1:  PR[GP1:91,2] = PR[GP1:90,2] + 26.774;
   1:L PR[91] 10mm/sec CNT100;
   1:  PR[GP1:91,1] = PR[GP1:90,1] + -67.229;
   1:  PR[GP1:91,2] = PR[GP1:90,2] + 21.599;
   1:L PR[91] 10mm/sec CNT100;
   1:  PR[GP1:91,1] = PR[GP1:90,1] + -71.366;
   1:  PR[GP1:91,2] = PR[GP1:90,2] + 14.920;
   1:L PR[91] 10mm/sec CNT100;
   1:  PR[GP1:91,1] = PR[GP1:90,1] + -73.727;
   1:  PR[GP1:91,2] = PR[GP1:90,2] + 8.074;
   1:L PR[91] 10mm/sec CNT100;
   1:  PR[GP1:91,1] = PR[GP1:90,1] + -74.537;
   1:  PR[GP1:91,2] = PR[GP1:90,2] + 0.787;
   1:L PR[91] 10mm/sec CNT100;
   1:  PR[GP1:91,1] = PR[GP1:90,1] + -74.638;
   1:  PR[GP1:91,2] = PR[GP1:90,2] + 0.256;
   1:L PR[91] 10mm/sec CNT100;
   1:  PR[GP1:91,1] = PR[GP1:90,1] + -73.834;
   1:  PR[GP1:91,2] = PR[GP1:90,2] + -6.976;
   1:L PR[91] 10mm/sec CNT100;
   1:  PR[GP1:91,1] = PR[GP1:90,1] + -73.735;
   1:  PR[GP1:91,2] = PR[GP1:90,2] + -7.493;
   1:L PR[91] 10mm/sec CNT100;
   1:  PR[GP1:91,1] = PR[GP1:90,1] + -71.365;
   1:  PR[GP1:91,2] = PR[GP1:90,2] + -14.362;
   1:L PR[91] 10mm/sec CNT100;
   1:  PR[GP1:91,1] = PR[GP1:90,1] + -67.524;
   1:  PR[GP1:91,2] = PR[GP1:90,2] + -20.577;
   1:L PR[91] 10mm/sec CNT100;
   1:  PR[GP1:91,1] = PR[GP1:90,1] + -67.231;
   1:  PR[GP1:91,2] = PR[GP1:90,2] + -21.039;
   1:L PR[91] 10mm/sec CNT100;
   1:  PR[GP1:91,1] = PR[GP1:90,1] + -62.171;
   1:  PR[GP1:91,2] = PR[GP1:90,2] + -26.204;
   1:L PR[91] 10mm/sec CNT100;
   1:  PR[GP1:91,1] = PR[GP1:90,1] + -56.033;
   1:  PR[GP1:91,2] = PR[GP1:90,2] + -30.176;
   1:L PR[91] 10mm/sec CNT100;
   1:  PR[GP1:91,1] = PR[GP1:90,1] + -55.573;
   1:  PR[GP1:91,2] = PR[GP1:90,2] + -30.512;
   1:L PR[91] 10mm/sec CNT100;
   1:  PR[GP1:91,1] = PR[GP1:90,1] + -48.797;
   1:  PR[GP1:91,2] = PR[GP1:90,2] + -33.007;
   1:L PR[91] 10mm/sec CNT100;
   1:  PR[GP1:91,1] = PR[GP1:90,1] + -48.177;
   1:  PR[GP1:91,2] = PR[GP1:90,2] + -33.168;
   1:L PR[91] 10mm/sec CNT100;
   1:  PR[GP1:91,1] = PR[GP1:90,1] + -41.043;
   1:  PR[GP1:91,2] = PR[GP1:90,2] + -34.110;
   1:L PR[91] 10mm/sec CNT100;
   1:  PR[GP1:91,1] = PR[GP1:90,1] + -33.849;
   1:  PR[GP1:91,2] = PR[GP1:90,2] + -33.460;
   1:L PR[91] 10mm/sec CNT100;
   1:  PR[GP1:91,1] = PR[GP1:90,1] + -33.160;
   1:  PR[GP1:91,2] = PR[GP1:90,2] + -33.377;
   1:L PR[91] 10mm/sec CNT100;
   1:  PR[GP1:91,1] = PR[GP1:90,1] + -26.373;
   1:  PR[GP1:91,2] = PR[GP1:90,2] + -31.191;
   1:L PR[91] 10mm/sec CNT100;
   1:  PR[GP1:91,1] = PR[GP1:90,1] + -20.171;
   1:  PR[GP1:91,2] = PR[GP1:90,2] + -27.532;
   1:L PR[91] 10mm/sec CNT100;
   1:  PR[GP1:91,1] = PR[GP1:90,1] + -19.505;
   1:  PR[GP1:91,2] = PR[GP1:90,2] + -27.174;
   1:L PR[91] 10mm/sec CNT100;
   1:  PR[GP1:91,1] = PR[GP1:90,1] + -14.336;
   1:  PR[GP1:91,2] = PR[GP1:90,2] + -22.316;
   1:L PR[91] 10mm/sec CNT100;
   1:  PR[GP1:91,1] = PR[GP1:90,1] + -13.779;
   1:  PR[GP1:91,2] = PR[GP1:90,2] + -21.655;
   1:L PR[91] 10mm/sec CNT100;
   1:  PR[GP1:91,1] = PR[GP1:90,1] + -9.819;
   1:  PR[GP1:91,2] = PR[GP1:90,2] + -15.802;
   1:L PR[91] 10mm/sec CNT100;
   1:  PR[GP1:91,1] = PR[GP1:90,1] + -7.234;
   1:  PR[GP1:91,2] = PR[GP1:90,2] + -9.204;
   1:L PR[91] 10mm/sec CNT100;
   1:  PR[GP1:91,1] = PR[GP1:90,1] + -6.942;
   1:  PR[GP1:91,2] = PR[GP1:90,2] + -8.345;
   1:L PR[91] 10mm/sec CNT100;
   1:  PR[GP1:91,1] = PR[GP1:90,1] + -5.885;
   1:  PR[GP1:91,2] = PR[GP1:90,2] + -1.442;
   1:L PR[91] 10mm/sec CNT100;
   1:  PR[GP1:91,1] = PR[GP1:90,1] + -6.031;
   1:  PR[GP1:91,2] = PR[GP1:90,2] + -0.737;
   1:L PR[91] 10mm/sec CNT100;
   1:  PR[GP1:91,1] = PR[GP1:90,1] + 5.283;
   1:  PR[GP1:91,2] = PR[GP1:90,2] + -0.738;
   1:L PR[91] 10mm/sec CNT100;
   1:  PR[GP1:91,1] = PR[GP1:90,1] + 5.916;
   1:  PR[GP1:91,2] = PR[GP1:90,2] + -5.183;
   1:  PR[GP1:91,3] = PR[GP1:90,3] + 9.455;
   1:L PR[91] 10mm/sec CNT100;
   1:  PR[GP1:91,1] = PR[GP1:90,1] + 6.295;
   1:  PR[GP1:91,2] = PR[GP1:90,2] + -7.974;
   1:L PR[91] 10mm/sec CNT100;
   1:  PR[GP1:91,1] = PR[GP1:90,1] + 8.636;
   1:  PR[GP1:91,2] = PR[GP1:90,2] + -13.949;
   1:L PR[91] 10mm/sec CNT100;
   1:  PR[GP1:91,1] = PR[GP1:90,1] + 9.298;
   1:  PR[GP1:91,2] = PR[GP1:90,2] + -15.893;
   1:L PR[91] 10mm/sec CNT100;
   1:  PR[GP1:91,1] = PR[GP1:90,1] + 12.891;
   1:  PR[GP1:91,2] = PR[GP1:90,2] + -21.202;
   1:L PR[91] 10mm/sec CNT100;
   1:  PR[GP1:91,1] = PR[GP1:90,1] + 14.126;
   1:  PR[GP1:91,2] = PR[GP1:90,2] + -22.668;
   1:L PR[91] 10mm/sec CNT100;
   1:  PR[GP1:91,1] = PR[GP1:90,1] + 18.869;
   1:  PR[GP1:91,2] = PR[GP1:90,2] + -27.126;
   1:L PR[91] 10mm/sec CNT100;
   1:  PR[GP1:91,1] = PR[GP1:90,1] + 24.496;
   1:  PR[GP1:91,2] = PR[GP1:90,2] + -30.446;
   1:L PR[91] 10mm/sec CNT100;
   1:  PR[GP1:91,1] = PR[GP1:90,1] + 26.069;
   1:  PR[GP1:91,2] = PR[GP1:90,2] + -31.295;
   1:L PR[91] 10mm/sec CNT100;
   1:  PR[GP1:91,1] = PR[GP1:90,1] + 32.342;
   1:  PR[GP1:91,2] = PR[GP1:90,2] + -33.315;
   1:L PR[91] 10mm/sec CNT100;
   1:  PR[GP1:91,1] = PR[GP1:90,1] + 38.969;
   1:  PR[GP1:91,2] = PR[GP1:90,2] + -33.914;
   1:L PR[91] 10mm/sec CNT100;
   1:  PR[GP1:91,1] = PR[GP1:90,1] + 40.606;
   1:  PR[GP1:91,2] = PR[GP1:90,2] + -34.109;
   1:L PR[91] 10mm/sec CNT100;
   1:  PR[GP1:91,1] = PR[GP1:90,1] + 47.242;
   1:  PR[GP1:91,2] = PR[GP1:90,2] + -33.232;
   1:L PR[91] 10mm/sec CNT100;
   1:  PR[GP1:91,1] = PR[GP1:90,1] + 48.635;
   1:  PR[GP1:91,2] = PR[GP1:90,2] + -32.871;
   1:L PR[91] 10mm/sec CNT100;
   1:  PR[GP1:91,1] = PR[GP1:90,1] + 55.004;
   1:  PR[GP1:91,2] = PR[GP1:90,2] + -30.526;
   1:L PR[91] 10mm/sec CNT100;
   1:  PR[GP1:91,1] = PR[GP1:90,1] + 60.713;
   1:  PR[GP1:91,2] = PR[GP1:90,2] + -26.833;
   1:L PR[91] 10mm/sec CNT100;
   1:  PR[GP1:91,1] = PR[GP1:90,1] + 61.800;
   1:  PR[GP1:91,2] = PR[GP1:90,2] + -26.042;
   1:L PR[91] 10mm/sec CNT100;
   1:  PR[GP1:91,1] = PR[GP1:90,1] + 66.572;
   1:  PR[GP1:91,2] = PR[GP1:90,2] + -21.170;
   1:L PR[91] 10mm/sec CNT100;
   1:  PR[GP1:91,1] = PR[GP1:90,1] + 70.187;
   1:  PR[GP1:91,2] = PR[GP1:90,2] + -15.323;
   1:L PR[91] 10mm/sec CNT100;
   1:  PR[GP1:91,1] = PR[GP1:90,1] + 70.868;
   1:  PR[GP1:91,2] = PR[GP1:90,2] + -14.246;
   1:L PR[91] 10mm/sec CNT100;
   1:  PR[GP1:91,1] = PR[GP1:90,1] + 73.097;
   1:  PR[GP1:91,2] = PR[GP1:90,2] + -7.787;
   1:L PR[91] 10mm/sec CNT100;
   1:  PR[GP1:91,1] = PR[GP1:90,1] + 73.862;
   1:  PR[GP1:91,2] = PR[GP1:90,2] + -0.903;
   1:L PR[91] 10mm/sec CNT100;
   1:  PR[GP1:91,1] = PR[GP1:90,1] + 74.090;
   1:  PR[GP1:91,2] = PR[GP1:90,2] + 0.302;
   1:L PR[91] 10mm/sec CNT100;
   1:  PR[GP1:91,1] = PR[GP1:90,1] + 73.329;
   1:  PR[GP1:91,2] = PR[GP1:90,2] + 7.146;
   1:L PR[91] 10mm/sec CNT100;
   1:  PR[GP1:91,1] = PR[GP1:90,1] + 73.104;
   1:  PR[GP1:91,2] = PR[GP1:90,2] + 8.322;
   1:L PR[91] 10mm/sec CNT100;
   1:  PR[GP1:91,1] = PR[GP1:90,1] + 70.867;
   1:  PR[GP1:91,2] = PR[GP1:90,2] + 14.807;
   1:L PR[91] 10mm/sec CNT100;
   1:  PR[GP1:91,1] = PR[GP1:90,1] + 67.240;
   1:  PR[GP1:91,2] = PR[GP1:90,2] + 20.676;
   1:L PR[91] 10mm/sec CNT100;
   1:  PR[GP1:91,1] = PR[GP1:90,1] + 66.575;
   1:  PR[GP1:91,2] = PR[GP1:90,2] + 21.725;
   1:L PR[91] 10mm/sec CNT100;
   1:  PR[GP1:91,1] = PR[GP1:90,1] + 61.811;
   1:  PR[GP1:91,2] = PR[GP1:90,2] + 26.588;
   1:L PR[91] 10mm/sec CNT100;
   1:  PR[GP1:91,1] = PR[GP1:90,1] + 56.028;
   1:  PR[GP1:91,2] = PR[GP1:90,2] + 30.329;
   1:L PR[91] 10mm/sec CNT100;
   1:  PR[GP1:91,1] = PR[GP1:90,1] + 54.987;
   1:  PR[GP1:91,2] = PR[GP1:90,2] + 31.091;
   1:L PR[91] 10mm/sec CNT100;
   1:  PR[GP1:91,1] = PR[GP1:90,1] + 48.635;
   1:  PR[GP1:91,2] = PR[GP1:90,2] + 33.429;
   1:L PR[91] 10mm/sec CNT100;
   1:  PR[GP1:91,1] = PR[GP1:90,1] + 47.243;
   1:  PR[GP1:91,2] = PR[GP1:90,2] + 33.790;
   1:L PR[91] 10mm/sec CNT100;
   1:  PR[GP1:91,1] = PR[GP1:90,1] + 40.597;
   1:  PR[GP1:91,2] = PR[GP1:90,2] + 34.668;
   1:L PR[91] 10mm/sec CNT100;
   1:  PR[GP1:91,1] = PR[GP1:90,1] + 33.894;
   1:  PR[GP1:91,2] = PR[GP1:90,2] + 34.063;
   1:L PR[91] 10mm/sec CNT100;
   1:  PR[GP1:91,1] = PR[GP1:90,1] + 32.351;
   1:  PR[GP1:91,2] = PR[GP1:90,2] + 33.876;
   1:L PR[91] 10mm/sec CNT100;
   1:  PR[GP1:91,1] = PR[GP1:90,1] + 26.080;
   1:  PR[GP1:91,2] = PR[GP1:90,2] + 31.856;
   1:L PR[91] 10mm/sec CNT100;
   1:  PR[GP1:91,1] = PR[GP1:90,1] + 20.346;
   1:  PR[GP1:91,2] = PR[GP1:90,2] + 28.473;
   1:L PR[91] 10mm/sec CNT100;
   1:  PR[GP1:91,1] = PR[GP1:90,1] + 18.860;
   1:  PR[GP1:91,2] = PR[GP1:90,2] + 27.676;
   1:L PR[91] 10mm/sec CNT100;
   1:  PR[GP1:91,1] = PR[GP1:90,1] + 14.126;
   1:  PR[GP1:91,2] = PR[GP1:90,2] + 23.226;
   1:L PR[91] 10mm/sec CNT100;
   1:  PR[GP1:91,1] = PR[GP1:90,1] + 12.891;
   1:  PR[GP1:91,2] = PR[GP1:90,2] + 21.760;
   1:L PR[91] 10mm/sec CNT100;
   1:  PR[GP1:91,1] = PR[GP1:90,1] + 9.290;
   1:  PR[GP1:91,2] = PR[GP1:90,2] + 16.439;
   1:L PR[91] 10mm/sec CNT100;
   1:  PR[GP1:91,1] = PR[GP1:90,1] + 6.940;
   1:  PR[GP1:91,2] = PR[GP1:90,2] + 10.441;
   1:L PR[91] 10mm/sec CNT100;
   1:  PR[GP1:91,1] = PR[GP1:90,1] + 6.295;
   1:  PR[GP1:91,2] = PR[GP1:90,2] + 8.540;
   1:L PR[91] 10mm/sec CNT100;
   1:  PR[GP1:91,1] = PR[GP1:90,1] + 5.339;
   1:  PR[GP1:91,2] = PR[GP1:90,2] + 2.298;
   1:L PR[91] 10mm/sec CNT100;
   1:  PR[GP1:91,1] = PR[GP1:90,1] + 5.507;
   1:  PR[GP1:91,2] = PR[GP1:90,2] + 1.495;
   1:L PR[91] 10mm/sec CNT100;
   1:  PR[GP1:91,1] = PR[GP1:90,1] + -5.813;
   1:  PR[GP1:91,2] = PR[GP1:90,2] + 1.494;
   1:L PR[91] 10mm/sec CNT100;
   1:  PR[GP1:91,1] = PR[GP1:90,1] + -6.442;
   1:  PR[GP1:91,2] = PR[GP1:90,2] + 5.741;
   1:L PR[91] 10mm/sec CNT100;
   1:  PR[GP1:91,1] = PR[GP1:90,1] + -6.821;
   1:  PR[GP1:91,2] = PR[GP1:90,2] + 8.532;
   1:L PR[91] 10mm/sec CNT100;
   1:  PR[GP1:91,1] = PR[GP1:90,1] + -9.162;
   1:  PR[GP1:91,2] = PR[GP1:90,2] + 14.507;
   1:L PR[91] 10mm/sec CNT100;
   1:  PR[GP1:91,1] = PR[GP1:90,1] + -9.825;
   1:  PR[GP1:91,2] = PR[GP1:90,2] + 16.452;
   1:L PR[91] 10mm/sec CNT100;
   1:  PR[GP1:91,1] = PR[GP1:90,1] + -13.418;
   1:  PR[GP1:91,2] = PR[GP1:90,2] + 21.762;
   1:L PR[91] 10mm/sec CNT100;
   1:  PR[GP1:91,1] = PR[GP1:90,1] + -14.653;
   1:  PR[GP1:91,2] = PR[GP1:90,2] + 23.226;
   1:L PR[91] 10mm/sec CNT100;
   1:  PR[GP1:91,1] = PR[GP1:90,1] + -19.396;
   1:  PR[GP1:91,2] = PR[GP1:90,2] + 27.685;
   1:L PR[91] 10mm/sec CNT100;
   1:  PR[GP1:91,1] = PR[GP1:90,1] + -25.023;
   1:  PR[GP1:91,2] = PR[GP1:90,2] + 31.005;
   1:L PR[91] 10mm/sec CNT100;
   1:  PR[GP1:91,1] = PR[GP1:90,1] + -26.596;
   1:  PR[GP1:91,2] = PR[GP1:90,2] + 31.853;
   1:L PR[91] 10mm/sec CNT100;
   1:  PR[GP1:91,1] = PR[GP1:90,1] + -32.869;
   1:  PR[GP1:91,2] = PR[GP1:90,2] + 33.873;
   1:L PR[91] 10mm/sec CNT100;
   1:  PR[GP1:91,1] = PR[GP1:90,1] + -39.496;
   1:  PR[GP1:91,2] = PR[GP1:90,2] + 34.472;
   1:L PR[91] 10mm/sec CNT100;
   1:  PR[GP1:91,1] = PR[GP1:90,1] + -41.133;
   1:  PR[GP1:91,2] = PR[GP1:90,2] + 34.667;
   1:L PR[91] 10mm/sec CNT100;
   1:  PR[GP1:91,1] = PR[GP1:90,1] + -47.769;
   1:  PR[GP1:91,2] = PR[GP1:90,2] + 33.790;
   1:L PR[91] 10mm/sec CNT100;
   1:  PR[GP1:91,1] = PR[GP1:90,1] + -49.162;
   1:  PR[GP1:91,2] = PR[GP1:90,2] + 33.429;
   1:L PR[91] 10mm/sec CNT100;
   1:  PR[GP1:91,1] = PR[GP1:90,1] + -55.530;
   1:  PR[GP1:91,2] = PR[GP1:90,2] + 31.084;
   1:L PR[91] 10mm/sec CNT100;
   1:  PR[GP1:91,1] = PR[GP1:90,1] + -61.239;
   1:  PR[GP1:91,2] = PR[GP1:90,2] + 27.391;
   1:L PR[91] 10mm/sec CNT100;
   1:  PR[GP1:91,1] = PR[GP1:90,1] + -62.326;
   1:  PR[GP1:91,2] = PR[GP1:90,2] + 26.600;
   1:L PR[91] 10mm/sec CNT100;
   1:  PR[GP1:91,1] = PR[GP1:90,1] + -67.099;
   1:  PR[GP1:91,2] = PR[GP1:90,2] + 21.727;
   1:L PR[91] 10mm/sec CNT100;
   1:  PR[GP1:91,1] = PR[GP1:90,1] + -70.713;
   1:  PR[GP1:91,2] = PR[GP1:90,2] + 15.881;
   1:L PR[91] 10mm/sec CNT100;
   1:  PR[GP1:91,1] = PR[GP1:90,1] + -71.395;
   1:  PR[GP1:91,2] = PR[GP1:90,2] + 14.804;
   1:L PR[91] 10mm/sec CNT100;
   1:  PR[GP1:91,1] = PR[GP1:90,1] + -73.623;
   1:  PR[GP1:91,2] = PR[GP1:90,2] + 8.345;
   1:L PR[91] 10mm/sec CNT100;
   1:  PR[GP1:91,1] = PR[GP1:90,1] + -74.388;
   1:  PR[GP1:91,2] = PR[GP1:90,2] + 1.461;
   1:L PR[91] 10mm/sec CNT100;
   1:  PR[GP1:91,1] = PR[GP1:90,1] + -74.617;
   1:  PR[GP1:91,2] = PR[GP1:90,2] + 0.256;
   1:L PR[91] 10mm/sec CNT100;
   1:  PR[GP1:91,1] = PR[GP1:90,1] + -73.856;
   1:  PR[GP1:91,2] = PR[GP1:90,2] + -6.588;
   1:L PR[91] 10mm/sec CNT100;
   1:  PR[GP1:91,1] = PR[GP1:90,1] + -73.631;
   1:  PR[GP1:91,2] = PR[GP1:90,2] + -7.764;
   1:L PR[91] 10mm/sec CNT100;
   1:  PR[GP1:91,1] = PR[GP1:90,1] + -71.394;
   1:  PR[GP1:91,2] = PR[GP1:90,2] + -14.249;
   1:L PR[91] 10mm/sec CNT100;
   1:  PR[GP1:91,1] = PR[GP1:90,1] + -67.766;
   1:  PR[GP1:91,2] = PR[GP1:90,2] + -20.118;
   1:L PR[91] 10mm/sec CNT100;
   1:  PR[GP1:91,1] = PR[GP1:90,1] + -67.101;
   1:  PR[GP1:91,2] = PR[GP1:90,2] + -21.167;
   1:L PR[91] 10mm/sec CNT100;
   1:  PR[GP1:91,1] = PR[GP1:90,1] + -62.338;
   1:  PR[GP1:91,2] = PR[GP1:90,2] + -26.030;
   1:L PR[91] 10mm/sec CNT100;
   1:  PR[GP1:91,1] = PR[GP1:90,1] + -56.555;
   1:  PR[GP1:91,2] = PR[GP1:90,2] + -29.771;
   1:L PR[91] 10mm/sec CNT100;
   1:  PR[GP1:91,1] = PR[GP1:90,1] + -55.514;
   1:  PR[GP1:91,2] = PR[GP1:90,2] + -30.532;
   1:L PR[91] 10mm/sec CNT100;
   1:  PR[GP1:91,1] = PR[GP1:90,1] + -49.162;
   1:  PR[GP1:91,2] = PR[GP1:90,2] + -32.871;
   1:L PR[91] 10mm/sec CNT100;
   1:  PR[GP1:91,1] = PR[GP1:90,1] + -47.769;
   1:  PR[GP1:91,2] = PR[GP1:90,2] + -33.232;
   1:L PR[91] 10mm/sec CNT100;
   1:  PR[GP1:91,1] = PR[GP1:90,1] + -41.124;
   1:  PR[GP1:91,2] = PR[GP1:90,2] + -34.110;
   1:L PR[91] 10mm/sec CNT100;
   1:  PR[GP1:91,1] = PR[GP1:90,1] + -34.421;
   1:  PR[GP1:91,2] = PR[GP1:90,2] + -33.504;
   1:L PR[91] 10mm/sec CNT100;
   1:  PR[GP1:91,1] = PR[GP1:90,1] + -32.878;
   1:  PR[GP1:91,2] = PR[GP1:90,2] + -33.318;
   1:L PR[91] 10mm/sec CNT100;
   1:  PR[GP1:91,1] = PR[GP1:90,1] + -26.607;
   1:  PR[GP1:91,2] = PR[GP1:90,2] + -31.299;
   1:L PR[91] 10mm/sec CNT100;
   1:  PR[GP1:91,1] = PR[GP1:90,1] + -20.873;
   1:  PR[GP1:91,2] = PR[GP1:90,2] + -27.915;
   1:L PR[91] 10mm/sec CNT100;
   1:  PR[GP1:91,1] = PR[GP1:90,1] + -19.387;
   1:  PR[GP1:91,2] = PR[GP1:90,2] + -27.118;
   1:L PR[91] 10mm/sec CNT100;
   1:  PR[GP1:91,1] = PR[GP1:90,1] + -14.653;
   1:  PR[GP1:91,2] = PR[GP1:90,2] + -22.668;
   1:L PR[91] 10mm/sec CNT100;
   1:  PR[GP1:91,1] = PR[GP1:90,1] + -13.418;
   1:  PR[GP1:91,2] = PR[GP1:90,2] + -21.204;
   1:L PR[91] 10mm/sec CNT100;
   1:  PR[GP1:91,1] = PR[GP1:90,1] + -9.817;
   1:  PR[GP1:91,2] = PR[GP1:90,2] + -15.883;
   1:L PR[91] 10mm/sec CNT100;
   1:  PR[GP1:91,1] = PR[GP1:90,1] + -7.467;
   1:  PR[GP1:91,2] = PR[GP1:90,2] + -9.884;
   1:L PR[91] 10mm/sec CNT100;
   1:  PR[GP1:91,1] = PR[GP1:90,1] + -6.821;
   1:  PR[GP1:91,2] = PR[GP1:90,2] + -7.982;
   1:L PR[91] 10mm/sec CNT100;
   1:  PR[GP1:91,1] = PR[GP1:90,1] + -5.866;
   1:  PR[GP1:91,2] = PR[GP1:90,2] + -1.740;
   1:L PR[91] 10mm/sec CNT100;
   1:  PR[GP1:91,1] = PR[GP1:90,1] + -6.033;
   1:  PR[GP1:91,2] = PR[GP1:90,2] + -0.937;
   1:L PR[91] 10mm/sec CNT100;
   1:  PR[GP1:91,1] = PR[GP1:90,1] + 5.286;
   1:  PR[GP1:91,2] = PR[GP1:90,2] + -0.936;
   1:L PR[91] 10mm/sec CNT100;
   1:  PR[GP1:91,1] = PR[GP1:90,1] + 5.590;
   1:  PR[GP1:91,2] = PR[GP1:90,2] + -3.304;
   1:  PR[GP1:91,3] = PR[GP1:90,3] + 10.065;
   1:L PR[91] 10mm/sec CNT100;
   1:  PR[GP1:91,1] = PR[GP1:90,1] + 6.174;
   1:  PR[GP1:91,2] = PR[GP1:90,2] + -7.611;
   1:L PR[91] 10mm/sec CNT100;
   1:  PR[GP1:91,1] = PR[GP1:90,1] + 8.272;
   1:  PR[GP1:91,2] = PR[GP1:90,2] + -12.965;
   1:L PR[91] 10mm/sec CNT100;
   1:  PR[GP1:91,1] = PR[GP1:90,1] + 9.297;
   1:  PR[GP1:91,2] = PR[GP1:90,2] + -15.973;
   1:L PR[91] 10mm/sec CNT100;
   1:  PR[GP1:91,1] = PR[GP1:90,1] + 12.529;
   1:  PR[GP1:91,2] = PR[GP1:90,2] + -20.750;
   1:L PR[91] 10mm/sec CNT100;
   1:  PR[GP1:91,1] = PR[GP1:90,1] + 14.443;
   1:  PR[GP1:91,2] = PR[GP1:90,2] + -23.020;
   1:L PR[91] 10mm/sec CNT100;
   1:  PR[GP1:91,1] = PR[GP1:90,1] + 18.751;
   1:  PR[GP1:91,2] = PR[GP1:90,2] + -27.070;
   1:L PR[91] 10mm/sec CNT100;
   1:  PR[GP1:91,1] = PR[GP1:90,1] + 23.864;
   1:  PR[GP1:91,2] = PR[GP1:90,2] + -30.087;
   1:L PR[91] 10mm/sec CNT100;
   1:  PR[GP1:91,1] = PR[GP1:90,1] + 26.303;
   1:  PR[GP1:91,2] = PR[GP1:90,2] + -31.402;
   1:L PR[91] 10mm/sec CNT100;
   1:  PR[GP1:91,1] = PR[GP1:90,1] + 32.060;
   1:  PR[GP1:91,2] = PR[GP1:90,2] + -33.256;
   1:L PR[91] 10mm/sec CNT100;
   1:  PR[GP1:91,1] = PR[GP1:90,1] + 38.146;
   1:  PR[GP1:91,2] = PR[GP1:90,2] + -33.806;
   1:L PR[91] 10mm/sec CNT100;
   1:  PR[GP1:91,1] = PR[GP1:90,1] + 40.686;
   1:  PR[GP1:91,2] = PR[GP1:90,2] + -34.109;
   1:L PR[91] 10mm/sec CNT100;
   1:  PR[GP1:91,1] = PR[GP1:90,1] + 46.835;
   1:  PR[GP1:91,2] = PR[GP1:90,2] + -33.297;
   1:L PR[91] 10mm/sec CNT100;
   1:  PR[GP1:91,1] = PR[GP1:90,1] + 49.000;
   1:  PR[GP1:91,2] = PR[GP1:90,2] + -32.736;
   1:L PR[91] 10mm/sec CNT100;
   1:  PR[GP1:91,1] = PR[GP1:90,1] + 54.945;
   1:  PR[GP1:91,2] = PR[GP1:90,2] + -30.547;
   1:L PR[91] 10mm/sec CNT100;
   1:  PR[GP1:91,1] = PR[GP1:90,1] + 60.274;
   1:  PR[GP1:91,2] = PR[GP1:90,2] + -27.099;
   1:L PR[91] 10mm/sec CNT100;
   1:  PR[GP1:91,1] = PR[GP1:90,1] + 61.966;
   1:  PR[GP1:91,2] = PR[GP1:90,2] + -25.867;
   1:L PR[91] 10mm/sec CNT100;
   1:  PR[GP1:91,1] = PR[GP1:90,1] + 66.443;
   1:  PR[GP1:91,2] = PR[GP1:90,2] + -21.297;
   1:L PR[91] 10mm/sec CNT100;
   1:  PR[GP1:91,1] = PR[GP1:90,1] + 69.834;
   1:  PR[GP1:91,2] = PR[GP1:90,2] + -15.810;
   1:L PR[91] 10mm/sec CNT100;
   1:  PR[GP1:91,1] = PR[GP1:90,1] + 70.897;
   1:  PR[GP1:91,2] = PR[GP1:90,2] + -14.133;
   1:L PR[91] 10mm/sec CNT100;
   1:  PR[GP1:91,1] = PR[GP1:90,1] + 72.992;
   1:  PR[GP1:91,2] = PR[GP1:90,2] + -8.058;
   1:L PR[91] 10mm/sec CNT100;
   1:  PR[GP1:91,1] = PR[GP1:90,1] + 73.713;
   1:  PR[GP1:91,2] = PR[GP1:90,2] + -1.578;
   1:L PR[91] 10mm/sec CNT100;
   1:  PR[GP1:91,1] = PR[GP1:90,1] + 74.069;
   1:  PR[GP1:91,2] = PR[GP1:90,2] + 0.302;
   1:L PR[91] 10mm/sec CNT100;
   1:  PR[GP1:91,1] = PR[GP1:90,1] + 73.351;
   1:  PR[GP1:91,2] = PR[GP1:90,2] + 6.758;
   1:L PR[91] 10mm/sec CNT100;
   1:  PR[GP1:91,1] = PR[GP1:90,1] + 73.000;
   1:  PR[GP1:91,2] = PR[GP1:90,2] + 8.593;
   1:L PR[91] 10mm/sec CNT100;
   1:  PR[GP1:91,1] = PR[GP1:90,1] + 70.895;
   1:  PR[GP1:91,2] = PR[GP1:90,2] + 14.694;
   1:L PR[91] 10mm/sec CNT100;
   1:  PR[GP1:91,1] = PR[GP1:90,1] + 67.481;
   1:  PR[GP1:91,2] = PR[GP1:90,2] + 20.218;
   1:L PR[91] 10mm/sec CNT100;
   1:  PR[GP1:91,1] = PR[GP1:90,1] + 66.445;
   1:  PR[GP1:91,2] = PR[GP1:90,2] + 21.853;
   1:L PR[91] 10mm/sec CNT100;
   1:  PR[GP1:91,1] = PR[GP1:90,1] + 61.978;
   1:  PR[GP1:91,2] = PR[GP1:90,2] + 26.414;
   1:L PR[91] 10mm/sec CNT100;
   1:  PR[GP1:91,1] = PR[GP1:90,1] + 56.550;
   1:  PR[GP1:91,2] = PR[GP1:90,2] + 29.925;
   1:L PR[91] 10mm/sec CNT100;
   1:  PR[GP1:91,1] = PR[GP1:90,1] + 54.928;
   1:  PR[GP1:91,2] = PR[GP1:90,2] + 31.111;
   1:L PR[91] 10mm/sec CNT100;
   1:  PR[GP1:91,1] = PR[GP1:90,1] + 49.000;
   1:  PR[GP1:91,2] = PR[GP1:90,2] + 33.294;
   1:L PR[91] 10mm/sec CNT100;
   1:  PR[GP1:91,1] = PR[GP1:90,1] + 46.835;
   1:  PR[GP1:91,2] = PR[GP1:90,2] + 33.855;
   1:L PR[91] 10mm/sec CNT100;
   1:  PR[GP1:91,1] = PR[GP1:90,1] + 40.678;
   1:  PR[GP1:91,2] = PR[GP1:90,2] + 34.668;
   1:L PR[91] 10mm/sec CNT100;
   1:  PR[GP1:91,1] = PR[GP1:90,1] + 34.465;
   1:  PR[GP1:91,2] = PR[GP1:90,2] + 34.107;
   1:L PR[91] 10mm/sec CNT100;
   1:  PR[GP1:91,1] = PR[GP1:90,1] + 32.068;
   1:  PR[GP1:91,2] = PR[GP1:90,2] + 33.817;
   1:L PR[91] 10mm/sec CNT100;
   1:  PR[GP1:91,1] = PR[GP1:90,1] + 26.314;
   1:  PR[GP1:91,2] = PR[GP1:90,2] + 31.964;
   1:L PR[91] 10mm/sec CNT100;
   1:  PR[GP1:91,1] = PR[GP1:90,1] + 21.047;
   1:  PR[GP1:91,2] = PR[GP1:90,2] + 28.857;
   1:L PR[91] 10mm/sec CNT100;
   1:  PR[GP1:91,1] = PR[GP1:90,1] + 18.742;
   1:  PR[GP1:91,2] = PR[GP1:90,2] + 27.620;
   1:L PR[91] 10mm/sec CNT100;
   1:  PR[GP1:91,1] = PR[GP1:90,1] + 14.443;
   1:  PR[GP1:91,2] = PR[GP1:90,2] + 23.578;
   1:L PR[91] 10mm/sec CNT100;
   1:  PR[GP1:91,1] = PR[GP1:90,1] + 12.529;
   1:  PR[GP1:91,2] = PR[GP1:90,2] + 21.308;
   1:L PR[91] 10mm/sec CNT100;
   1:  PR[GP1:91,1] = PR[GP1:90,1] + 9.289;
   1:  PR[GP1:91,2] = PR[GP1:90,2] + 16.520;
   1:L PR[91] 10mm/sec CNT100;
   1:  PR[GP1:91,1] = PR[GP1:90,1] + 7.173;
   1:  PR[GP1:91,2] = PR[GP1:90,2] + 11.119;
   1:L PR[91] 10mm/sec CNT100;
   1:  PR[GP1:91,1] = PR[GP1:90,1] + 6.174;
   1:  PR[GP1:91,2] = PR[GP1:90,2] + 8.177;
   1:L PR[91] 10mm/sec CNT100;
   1:  PR[GP1:91,1] = PR[GP1:90,1] + 5.322;
   1:  PR[GP1:91,2] = PR[GP1:90,2] + 2.610;
   1:L PR[91] 10mm/sec CNT100;
   1:  PR[GP1:91,1] = PR[GP1:90,1] + 5.535;
   1:  PR[GP1:91,2] = PR[GP1:90,2] + 1.775;
   1:L PR[91] 10mm/sec CNT100;
   1:  PR[GP1:91,1] = PR[GP1:90,1] + -5.807;
   1:  PR[GP1:91,2] = PR[GP1:90,2] + 1.773;
   1:L PR[91] 10mm/sec CNT100;
   1:  PR[GP1:91,1] = PR[GP1:90,1] + -6.116;
   1:  PR[GP1:91,2] = PR[GP1:90,2] + 3.862;
   1:L PR[91] 10mm/sec CNT100;
   1:  PR[GP1:91,1] = PR[GP1:90,1] + -6.701;
   1:  PR[GP1:91,2] = PR[GP1:90,2] + 8.169;
   1:L PR[91] 10mm/sec CNT100;
   1:  PR[GP1:91,1] = PR[GP1:90,1] + -8.798;
   1:  PR[GP1:91,2] = PR[GP1:90,2] + 13.523;
   1:L PR[91] 10mm/sec CNT100;
   1:  PR[GP1:91,1] = PR[GP1:90,1] + -9.824;
   1:  PR[GP1:91,2] = PR[GP1:90,2] + 16.533;
   1:L PR[91] 10mm/sec CNT100;
   1:  PR[GP1:91,1] = PR[GP1:90,1] + -13.056;
   1:  PR[GP1:91,2] = PR[GP1:90,2] + 21.310;
   1:L PR[91] 10mm/sec CNT100;
   1:  PR[GP1:91,1] = PR[GP1:90,1] + -14.970;
   1:  PR[GP1:91,2] = PR[GP1:90,2] + 23.579;
   1:L PR[91] 10mm/sec CNT100;
   1:  PR[GP1:91,1] = PR[GP1:90,1] + -19.278;
   1:  PR[GP1:91,2] = PR[GP1:90,2] + 27.629;
   1:L PR[91] 10mm/sec CNT100;
   1:  PR[GP1:91,1] = PR[GP1:90,1] + -24.392;
   1:  PR[GP1:91,2] = PR[GP1:90,2] + 30.646;
   1:L PR[91] 10mm/sec CNT100;
   1:  PR[GP1:91,1] = PR[GP1:90,1] + -26.830;
   1:  PR[GP1:91,2] = PR[GP1:90,2] + 31.961;
   1:L PR[91] 10mm/sec CNT100;
   1:  PR[GP1:91,1] = PR[GP1:90,1] + -32.587;
   1:  PR[GP1:91,2] = PR[GP1:90,2] + 33.815;
   1:L PR[91] 10mm/sec CNT100;
   1:  PR[GP1:91,1] = PR[GP1:90,1] + -38.674;
   1:  PR[GP1:91,2] = PR[GP1:90,2] + 34.365;
   1:L PR[91] 10mm/sec CNT100;
   1:  PR[GP1:91,1] = PR[GP1:90,1] + -41.213;
   1:  PR[GP1:91,2] = PR[GP1:90,2] + 34.667;
   1:L PR[91] 10mm/sec CNT100;
   1:  PR[GP1:91,1] = PR[GP1:90,1] + -47.362;
   1:  PR[GP1:91,2] = PR[GP1:90,2] + 33.855;
   1:L PR[91] 10mm/sec CNT100;
   1:  PR[GP1:91,1] = PR[GP1:90,1] + -49.527;
   1:  PR[GP1:91,2] = PR[GP1:90,2] + 33.293;
   1:L PR[91] 10mm/sec CNT100;
   1:  PR[GP1:91,1] = PR[GP1:90,1] + -55.471;
   1:  PR[GP1:91,2] = PR[GP1:90,2] + 31.105;
   1:L PR[91] 10mm/sec CNT100;
   1:  PR[GP1:91,1] = PR[GP1:90,1] + -60.801;
   1:  PR[GP1:91,2] = PR[GP1:90,2] + 27.657;
   1:L PR[91] 10mm/sec CNT100;
   1:  PR[GP1:91,1] = PR[GP1:90,1] + -62.493;
   1:  PR[GP1:91,2] = PR[GP1:90,2] + 26.425;
   1:L PR[91] 10mm/sec CNT100;
   1:  PR[GP1:91,1] = PR[GP1:90,1] + -66.969;
   1:  PR[GP1:91,2] = PR[GP1:90,2] + 21.855;
   1:L PR[91] 10mm/sec CNT100;
   1:  PR[GP1:91,1] = PR[GP1:90,1] + -70.361;
   1:  PR[GP1:91,2] = PR[GP1:90,2] + 16.368;
   1:L PR[91] 10mm/sec CNT100;
   1:  PR[GP1:91,1] = PR[GP1:90,1] + -71.423;
   1:  PR[GP1:91,2] = PR[GP1:90,2] + 14.691;
   1:L PR[91] 10mm/sec CNT100;
   1:  PR[GP1:91,1] = PR[GP1:90,1] + -73.519;
   1:  PR[GP1:91,2] = PR[GP1:90,2] + 8.615;
   1:L PR[91] 10mm/sec CNT100;
   1:  PR[GP1:91,1] = PR[GP1:90,1] + -74.239;
   1:  PR[GP1:91,2] = PR[GP1:90,2] + 2.135;
   1:L PR[91] 10mm/sec CNT100;
   1:  PR[GP1:91,1] = PR[GP1:90,1] + -74.595;
   1:  PR[GP1:91,2] = PR[GP1:90,2] + 0.256;
   1:L PR[91] 10mm/sec CNT100;
   1:  PR[GP1:91,1] = PR[GP1:90,1] + -73.877;
   1:  PR[GP1:91,2] = PR[GP1:90,2] + -6.200;
   1:L PR[91] 10mm/sec CNT100;
   1:  PR[GP1:91,1] = PR[GP1:90,1] + -73.526;
   1:  PR[GP1:91,2] = PR[GP1:90,2] + -8.035;
   1:L PR[91] 10mm/sec CNT100;
   1:  PR[GP1:91,1] = PR[GP1:90,1] + -71.422;
   1:  PR[GP1:91,2] = PR[GP1:90,2] + -14.136;
   1:L PR[91] 10mm/sec CNT100;
   1:  PR[GP1:91,1] = PR[GP1:90,1] + -68.008;
   1:  PR[GP1:91,2] = PR[GP1:90,2] + -19.659;
   1:L PR[91] 10mm/sec CNT100;
   1:  PR[GP1:91,1] = PR[GP1:90,1] + -66.972;
   1:  PR[GP1:91,2] = PR[GP1:90,2] + -21.295;
   1:L PR[91] 10mm/sec CNT100;
   1:  PR[GP1:91,1] = PR[GP1:90,1] + -62.504;
   1:  PR[GP1:91,2] = PR[GP1:90,2] + -25.855;
   1:L PR[91] 10mm/sec CNT100;
   1:  PR[GP1:91,1] = PR[GP1:90,1] + -57.077;
   1:  PR[GP1:91,2] = PR[GP1:90,2] + -29.367;
   1:L PR[91] 10mm/sec CNT100;
   1:  PR[GP1:91,1] = PR[GP1:90,1] + -55.455;
   1:  PR[GP1:91,2] = PR[GP1:90,2] + -30.553;
   1:L PR[91] 10mm/sec CNT100;
   1:  PR[GP1:91,1] = PR[GP1:90,1] + -49.527;
   1:  PR[GP1:91,2] = PR[GP1:90,2] + -32.735;
   1:L PR[91] 10mm/sec CNT100;
   1:  PR[GP1:91,1] = PR[GP1:90,1] + -47.362;
   1:  PR[GP1:91,2] = PR[GP1:90,2] + -33.297;
   1:L PR[91] 10mm/sec CNT100;
   1:  PR[GP1:91,1] = PR[GP1:90,1] + -41.205;
   1:  PR[GP1:91,2] = PR[GP1:90,2] + -34.110;
   1:L PR[91] 10mm/sec CNT100;
   1:  PR[GP1:91,1] = PR[GP1:90,1] + -34.992;
   1:  PR[GP1:91,2] = PR[GP1:90,2] + -33.549;
   1:L PR[91] 10mm/sec CNT100;
   1:  PR[GP1:91,1] = PR[GP1:90,1] + -32.596;
   1:  PR[GP1:91,2] = PR[GP1:90,2] + -33.260;
   1:L PR[91] 10mm/sec CNT100;
   1:  PR[GP1:91,1] = PR[GP1:90,1] + -26.841;
   1:  PR[GP1:91,2] = PR[GP1:90,2] + -31.406;
   1:L PR[91] 10mm/sec CNT100;
   1:  PR[GP1:91,1] = PR[GP1:90,1] + -21.574;
   1:  PR[GP1:91,2] = PR[GP1:90,2] + -28.299;
   1:L PR[91] 10mm/sec CNT100;
   1:  PR[GP1:91,1] = PR[GP1:90,1] + -19.269;
   1:  PR[GP1:91,2] = PR[GP1:90,2] + -27.062;
   1:L PR[91] 10mm/sec CNT100;
   1:  PR[GP1:91,1] = PR[GP1:90,1] + -14.970;
   1:  PR[GP1:91,2] = PR[GP1:90,2] + -23.021;
   1:L PR[91] 10mm/sec CNT100;
   1:  PR[GP1:91,1] = PR[GP1:90,1] + -13.056;
   1:  PR[GP1:91,2] = PR[GP1:90,2] + -20.752;
   1:L PR[91] 10mm/sec CNT100;
   1:  PR[GP1:91,1] = PR[GP1:90,1] + -9.816;
   1:  PR[GP1:91,2] = PR[GP1:90,2] + -15.964;
   1:L PR[91] 10mm/sec CNT100;
   1:  PR[GP1:91,1] = PR[GP1:90,1] + -7.701;
   1:  PR[GP1:91,2] = PR[GP1:90,2] + -10.563;
   1:L PR[91] 10mm/sec CNT100;
   1:  PR[GP1:91,1] = PR[GP1:90,1] + -6.701;
   1:  PR[GP1:91,2] = PR[GP1:90,2] + -7.619;
   1:L PR[91] 10mm/sec CNT100;
   1:  PR[GP1:91,1] = PR[GP1:90,1] + -5.848;
   1:  PR[GP1:91,2] = PR[GP1:90,2] + -2.051;
   1:L PR[91] 10mm/sec CNT100;
   1:  PR[GP1:91,1] = PR[GP1:90,1] + -6.061;
   1:  PR[GP1:91,2] = PR[GP1:90,2] + -1.217;
   1:L PR[91] 10mm/sec CNT100;
   1:  PR[GP1:91,1] = PR[GP1:90,1] + 5.280;
   1:  PR[GP1:91,2] = PR[GP1:90,2] + -1.215;
   1:L PR[91] 10mm/sec CNT100;
   1:  PR[GP1:91,1] = PR[GP1:90,1] + 6.054;
   1:  PR[GP1:91,2] = PR[GP1:90,2] + -7.249;
   1:  PR[GP1:91,3] = PR[GP1:90,3] + 10.675;
   1:L PR[91] 10mm/sec CNT100;
   1:  PR[GP1:91,1] = PR[GP1:90,1] + 7.907;
   1:  PR[GP1:91,2] = PR[GP1:90,2] + -11.981;
   1:L PR[91] 10mm/sec CNT100;
   1:  PR[GP1:91,1] = PR[GP1:90,1] + 9.295;
   1:  PR[GP1:91,2] = PR[GP1:90,2] + -16.053;
   1:L PR[91] 10mm/sec CNT100;
   1:  PR[GP1:91,1] = PR[GP1:90,1] + 12.167;
   1:  PR[GP1:91,2] = PR[GP1:90,2] + -20.298;
   1:L PR[91] 10mm/sec CNT100;
   1:  PR[GP1:91,1] = PR[GP1:90,1] + 14.759;
   1:  PR[GP1:91,2] = PR[GP1:90,2] + -23.372;
   1:L PR[91] 10mm/sec CNT100;
   1:  PR[GP1:91,1] = PR[GP1:90,1] + 18.633;
   1:  PR[GP1:91,2] = PR[GP1:90,2] + -27.014;
   1:L PR[91] 10mm/sec CNT100;
   1:  PR[GP1:91,1] = PR[GP1:90,1] + 23.232;
   1:  PR[GP1:91,2] = PR[GP1:90,2] + -29.728;
   1:L PR[91] 10mm/sec CNT100;
   1:  PR[GP1:91,1] = PR[GP1:90,1] + 26.537;
   1:  PR[GP1:91,2] = PR[GP1:90,2] + -31.510;
   1:L PR[91] 10mm/sec CNT100;
   1:  PR[GP1:91,1] = PR[GP1:90,1] + 31.777;
   1:  PR[GP1:91,2] = PR[GP1:90,2] + -33.198;
   1:L PR[91] 10mm/sec CNT100;
   1:  PR[GP1:91,1] = PR[GP1:90,1] + 37.323;
   1:  PR[GP1:91,2] = PR[GP1:90,2] + -33.699;
   1:L PR[91] 10mm/sec CNT100;
   1:  PR[GP1:91,1] = PR[GP1:90,1] + 40.767;
   1:  PR[GP1:91,2] = PR[GP1:90,2] + -34.109;
   1:L PR[91] 10mm/sec CNT100;
   1:  PR[GP1:91,1] = PR[GP1:90,1] + 46.427;
   1:  PR[GP1:91,2] = PR[GP1:90,2] + -33.362;
   1:L PR[91] 10mm/sec CNT100;
   1:  PR[GP1:91,1] = PR[GP1:90,1] + 49.366;
   1:  PR[GP1:91,2] = PR[GP1:90,2] + -32.600;
   1:L PR[91] 10mm/sec CNT100;
   1:  PR[GP1:91,1] = PR[GP1:90,1] + 54.885;
   1:  PR[GP1:91,2] = PR[GP1:90,2] + -30.567;
   1:L PR[91] 10mm/sec CNT100;
   1:  PR[GP1:91,1] = PR[GP1:90,1] + 59.835;
   1:  PR[GP1:91,2] = PR[GP1:90,2] + -27.365;
   1:L PR[91] 10mm/sec CNT100;
   1:  PR[GP1:91,1] = PR[GP1:90,1] + 62.132;
   1:  PR[GP1:91,2] = PR[GP1:90,2] + -25.693;
   1:L PR[91] 10mm/sec CNT100;
   1:  PR[GP1:91,1] = PR[GP1:90,1] + 66.313;
   1:  PR[GP1:91,2] = PR[GP1:90,2] + -21.425;
   1:L PR[91] 10mm/sec CNT100;
   1:  PR[GP1:91,1] = PR[GP1:90,1] + 69.482;
   1:  PR[GP1:91,2] = PR[GP1:90,2] + -16.298;
   1:L PR[91] 10mm/sec CNT100;
   1:  PR[GP1:91,1] = PR[GP1:90,1] + 70.925;
   1:  PR[GP1:91,2] = PR[GP1:90,2] + -14.020;
   1:L PR[91] 10mm/sec CNT100;
   1:  PR[GP1:91,1] = PR[GP1:90,1] + 72.888;
   1:  PR[GP1:91,2] = PR[GP1:90,2] + -8.329;
   1:L PR[91] 10mm/sec CNT100;
   1:  PR[GP1:91,1] = PR[GP1:90,1] + 73.564;
   1:  PR[GP1:91,2] = PR[GP1:90,2] + -2.252;
   1:L PR[91] 10mm/sec CNT100;
   1:  PR[GP1:91,1] = PR[GP1:90,1] + 74.048;
   1:  PR[GP1:91,2] = PR[GP1:90,2] + 0.302;
   1:L PR[91] 10mm/sec CNT100;
   1:  PR[GP1:91,1] = PR[GP1:90,1] + 73.373;
   1:  PR[GP1:91,2] = PR[GP1:90,2] + 6.370;
   1:L PR[91] 10mm/sec CNT100;
   1:  PR[GP1:91,1] = PR[GP1:90,1] + 72.896;
   1:  PR[GP1:91,2] = PR[GP1:90,2] + 8.864;
   1:L PR[91] 10mm/sec CNT100;
   1:  PR[GP1:91,1] = PR[GP1:90,1] + 70.924;
   1:  PR[GP1:91,2] = PR[GP1:90,2] + 14.581;
   1:L PR[91] 10mm/sec CNT100;
   1:  PR[GP1:91,1] = PR[GP1:90,1] + 67.723;
   1:  PR[GP1:91,2] = PR[GP1:90,2] + 19.760;
   1:L PR[91] 10mm/sec CNT100;
   1:  PR[GP1:91,1] = PR[GP1:90,1] + 66.315;
   1:  PR[GP1:91,2] = PR[GP1:90,2] + 21.981;
   1:L PR[91] 10mm/sec CNT100;
   1:  PR[GP1:91,1] = PR[GP1:90,1] + 62.144;
   1:  PR[GP1:91,2] = PR[GP1:90,2] + 26.239;
   1:L PR[91] 10mm/sec CNT100;
   1:  PR[GP1:91,1] = PR[GP1:90,1] + 57.072;
   1:  PR[GP1:91,2] = PR[GP1:90,2] + 29.521;
   1:L PR[91] 10mm/sec CNT100;
   1:  PR[GP1:91,1] = PR[GP1:90,1] + 54.869;
   1:  PR[GP1:91,2] = PR[GP1:90,2] + 31.131;
   1:L PR[91] 10mm/sec CNT100;
   1:  PR[GP1:91,1] = PR[GP1:90,1] + 49.366;
   1:  PR[GP1:91,2] = PR[GP1:90,2] + 33.158;
   1:L PR[91] 10mm/sec CNT100;
   1:  PR[GP1:91,1] = PR[GP1:90,1] + 46.427;
   1:  PR[GP1:91,2] = PR[GP1:90,2] + 33.920;
   1:L PR[91] 10mm/sec CNT100;
   1:  PR[GP1:91,1] = PR[GP1:90,1] + 40.758;
   1:  PR[GP1:91,2] = PR[GP1:90,2] + 34.669;
   1:L PR[91] 10mm/sec CNT100;
   1:  PR[GP1:91,1] = PR[GP1:90,1] + 35.036;
   1:  PR[GP1:91,2] = PR[GP1:90,2] + 34.151;
   1:L PR[91] 10mm/sec CNT100;
   1:  PR[GP1:91,1] = PR[GP1:90,1] + 31.786;
   1:  PR[GP1:91,2] = PR[GP1:90,2] + 33.759;
   1:L PR[91] 10mm/sec CNT100;
   1:  PR[GP1:91,1] = PR[GP1:90,1] + 26.548;
   1:  PR[GP1:91,2] = PR[GP1:90,2] + 32.072;
   1:L PR[91] 10mm/sec CNT100;
   1:  PR[GP1:91,1] = PR[GP1:90,1] + 21.748;
   1:  PR[GP1:91,2] = PR[GP1:90,2] + 29.240;
   1:L PR[91] 10mm/sec CNT100;
   1:  PR[GP1:91,1] = PR[GP1:90,1] + 18.624;
   1:  PR[GP1:91,2] = PR[GP1:90,2] + 27.563;
   1:L PR[91] 10mm/sec CNT100;
   1:  PR[GP1:91,1] = PR[GP1:90,1] + 14.759;
   1:  PR[GP1:91,2] = PR[GP1:90,2] + 23.930;
   1:L PR[91] 10mm/sec CNT100;
   1:  PR[GP1:91,1] = PR[GP1:90,1] + 12.167;
   1:  PR[GP1:91,2] = PR[GP1:90,2] + 20.856;
   1:L PR[91] 10mm/sec CNT100;
   1:  PR[GP1:91,1] = PR[GP1:90,1] + 9.288;
   1:  PR[GP1:91,2] = PR[GP1:90,2] + 16.600;
   1:L PR[91] 10mm/sec CNT100;
   1:  PR[GP1:91,1] = PR[GP1:90,1] + 7.406;
   1:  PR[GP1:91,2] = PR[GP1:90,2] + 11.798;
   1:L PR[91] 10mm/sec CNT100;
   1:  PR[GP1:91,1] = PR[GP1:90,1] + 6.054;
   1:  PR[GP1:91,2] = PR[GP1:90,2] + 7.814;
   1:L PR[91] 10mm/sec CNT100;
   1:  PR[GP1:91,1] = PR[GP1:90,1] + 5.304;
   1:  PR[GP1:91,2] = PR[GP1:90,2] + 2.916;
   1:L PR[91] 10mm/sec CNT100;
   1:  PR[GP1:91,1] = PR[GP1:90,1] + 5.545;
   1:  PR[GP1:91,2] = PR[GP1:90,2] + 2.067;
   1:L PR[91] 10mm/sec CNT100;
   1:  PR[GP1:91,1] = PR[GP1:90,1] + -5.801;
   1:L PR[91] 10mm/sec CNT100;
   1:  PR[GP1:91,1] = PR[GP1:90,1] + -6.580;
   1:  PR[GP1:91,2] = PR[GP1:90,2] + 7.807;
   1:L PR[91] 10mm/sec CNT100;
   1:  PR[GP1:91,1] = PR[GP1:90,1] + -8.434;
   1:  PR[GP1:91,2] = PR[GP1:90,2] + 12.539;
   1:L PR[91] 10mm/sec CNT100;
   1:  PR[GP1:91,1] = PR[GP1:90,1] + -9.823;
   1:  PR[GP1:91,2] = PR[GP1:90,2] + 16.614;
   1:L PR[91] 10mm/sec CNT100;
   1:  PR[GP1:91,1] = PR[GP1:90,1] + -12.695;
   1:  PR[GP1:91,2] = PR[GP1:90,2] + 20.859;
   1:L PR[91] 10mm/sec CNT100;
   1:  PR[GP1:91,1] = PR[GP1:90,1] + -15.286;
   1:  PR[GP1:91,2] = PR[GP1:90,2] + 23.931;
   1:L PR[91] 10mm/sec CNT100;
   1:  PR[GP1:91,1] = PR[GP1:90,1] + -19.161;
   1:  PR[GP1:91,2] = PR[GP1:90,2] + 27.573;
   1:L PR[91] 10mm/sec CNT100;
   1:  PR[GP1:91,1] = PR[GP1:90,1] + -23.760;
   1:  PR[GP1:91,2] = PR[GP1:90,2] + 30.287;
   1:L PR[91] 10mm/sec CNT100;
   1:  PR[GP1:91,1] = PR[GP1:90,1] + -27.064;
   1:  PR[GP1:91,2] = PR[GP1:90,2] + 32.069;
   1:L PR[91] 10mm/sec CNT100;
   1:  PR[GP1:91,1] = PR[GP1:90,1] + -32.305;
   1:  PR[GP1:91,2] = PR[GP1:90,2] + 33.756;
   1:L PR[91] 10mm/sec CNT100;
   1:  PR[GP1:91,1] = PR[GP1:90,1] + -37.851;
   1:  PR[GP1:91,2] = PR[GP1:90,2] + 34.258;
   1:L PR[91] 10mm/sec CNT100;
   1:  PR[GP1:91,1] = PR[GP1:90,1] + -41.294;
   1:  PR[GP1:91,2] = PR[GP1:90,2] + 34.667;
   1:L PR[91] 10mm/sec CNT100;
   1:  PR[GP1:91,1] = PR[GP1:90,1] + -46.954;
   1:  PR[GP1:91,2] = PR[GP1:90,2] + 33.920;
   1:L PR[91] 10mm/sec CNT100;
   1:  PR[GP1:91,1] = PR[GP1:90,1] + -49.893;
   1:  PR[GP1:91,2] = PR[GP1:90,2] + 33.157;
   1:L PR[91] 10mm/sec CNT100;
   1:  PR[GP1:91,1] = PR[GP1:90,1] + -55.412;
   1:  PR[GP1:91,2] = PR[GP1:90,2] + 31.125;
   1:L PR[91] 10mm/sec CNT100;
   1:  PR[GP1:91,1] = PR[GP1:90,1] + -60.362;
   1:  PR[GP1:91,2] = PR[GP1:90,2] + 27.923;
   1:L PR[91] 10mm/sec CNT100;
   1:  PR[GP1:91,1] = PR[GP1:90,1] + -62.659;
   1:  PR[GP1:91,2] = PR[GP1:90,2] + 26.251;
   1:L PR[91] 10mm/sec CNT100;
   1:  PR[GP1:91,1] = PR[GP1:90,1] + -66.840;
   1:  PR[GP1:91,2] = PR[GP1:90,2] + 21.983;
   1:L PR[91] 10mm/sec CNT100;
   1:  PR[GP1:91,1] = PR[GP1:90,1] + -70.009;
   1:  PR[GP1:91,2] = PR[GP1:90,2] + 16.856;
   1:L PR[91] 10mm/sec CNT100;
   1:  PR[GP1:91,1] = PR[GP1:90,1] + -71.451;
   1:  PR[GP1:91,2] = PR[GP1:90,2] + 14.578;
   1:L PR[91] 10mm/sec CNT100;
   1:  PR[GP1:91,1] = PR[GP1:90,1] + -73.415;
   1:  PR[GP1:91,2] = PR[GP1:90,2] + 8.886;
   1:L PR[91] 10mm/sec CNT100;
   1:  PR[GP1:91,1] = PR[GP1:90,1] + -74.090;
   1:  PR[GP1:91,2] = PR[GP1:90,2] + 2.810;
   1:L PR[91] 10mm/sec CNT100;
   1:  PR[GP1:91,1] = PR[GP1:90,1] + -74.574;
   1:  PR[GP1:91,2] = PR[GP1:90,2] + 0.256;
   1:L PR[91] 10mm/sec CNT100;
   1:  PR[GP1:91,1] = PR[GP1:90,1] + -73.899;
   1:  PR[GP1:91,2] = PR[GP1:90,2] + -5.812;
   1:L PR[91] 10mm/sec CNT100;
   1:  PR[GP1:91,1] = PR[GP1:90,1] + -73.422;
   1:  PR[GP1:91,2] = PR[GP1:90,2] + -8.305;
   1:L PR[91] 10mm/sec CNT100;
   1:  PR[GP1:91,1] = PR[GP1:90,1] + -71.450;
   1:  PR[GP1:91,2] = PR[GP1:90,2] + -14.023;
   1:L PR[91] 10mm/sec CNT100;
   1:  PR[GP1:91,1] = PR[GP1:90,1] + -68.250;
   1:  PR[GP1:91,2] = PR[GP1:90,2] + -19.200;
   1:L PR[91] 10mm/sec CNT100;
   1:  PR[GP1:91,1] = PR[GP1:90,1] + -66.842;
   1:  PR[GP1:91,2] = PR[GP1:90,2] + -21.423;
   1:L PR[91] 10mm/sec CNT100;
   1:  PR[GP1:91,1] = PR[GP1:90,1] + -62.671;
   1:  PR[GP1:91,2] = PR[GP1:90,2] + -25.681;
   1:L PR[91] 10mm/sec CNT100;
   1:  PR[GP1:91,1] = PR[GP1:90,1] + -57.598;
   1:  PR[GP1:91,2] = PR[GP1:90,2] + -28.963;
   1:L PR[91] 10mm/sec CNT100;
   1:  PR[GP1:91,1] = PR[GP1:90,1] + -55.396;
   1:  PR[GP1:91,2] = PR[GP1:90,2] + -30.573;
   1:L PR[91] 10mm/sec CNT100;
   1:  PR[GP1:91,1] = PR[GP1:90,1] + -49.893;
   1:  PR[GP1:91,2] = PR[GP1:90,2] + -32.599;
   1:L PR[91] 10mm/sec CNT100;
   1:  PR[GP1:91,1] = PR[GP1:90,1] + -46.954;
   1:  PR[GP1:91,2] = PR[GP1:90,2] + -33.362;
   1:L PR[91] 10mm/sec CNT100;
   1:  PR[GP1:91,1] = PR[GP1:90,1] + -41.286;
   1:  PR[GP1:91,2] = PR[GP1:90,2] + -34.110;
   1:L PR[91] 10mm/sec CNT100;
   1:  PR[GP1:91,1] = PR[GP1:90,1] + -35.563;
   1:  PR[GP1:91,2] = PR[GP1:90,2] + -33.593;
   1:L PR[91] 10mm/sec CNT100;
   1:  PR[GP1:91,1] = PR[GP1:90,1] + -32.313;
   1:  PR[GP1:91,2] = PR[GP1:90,2] + -33.201;
   1:L PR[91] 10mm/sec CNT100;
   1:  PR[GP1:91,1] = PR[GP1:90,1] + -27.076;
   1:  PR[GP1:91,2] = PR[GP1:90,2] + -31.514;
   1:L PR[91] 10mm/sec CNT100;
   1:  PR[GP1:91,1] = PR[GP1:90,1] + -22.276;
   1:  PR[GP1:91,2] = PR[GP1:90,2] + -28.682;
   1:L PR[91] 10mm/sec CNT100;
   1:  PR[GP1:91,1] = PR[GP1:90,1] + -19.152;
   1:  PR[GP1:91,2] = PR[GP1:90,2] + -27.006;
   1:L PR[91] 10mm/sec CNT100;
   1:  PR[GP1:91,1] = PR[GP1:90,1] + -15.286;
   1:  PR[GP1:91,2] = PR[GP1:90,2] + -23.373;
   1:L PR[91] 10mm/sec CNT100;
   1:  PR[GP1:91,1] = PR[GP1:90,1] + -12.695;
   1:  PR[GP1:91,2] = PR[GP1:90,2] + -20.301;
   1:L PR[91] 10mm/sec CNT100;
   1:  PR[GP1:91,1] = PR[GP1:90,1] + -9.815;
   1:  PR[GP1:91,2] = PR[GP1:90,2] + -16.045;
   1:L PR[91] 10mm/sec CNT100;
   1:  PR[GP1:91,1] = PR[GP1:90,1] + -7.934;
   1:  PR[GP1:91,2] = PR[GP1:90,2] + -11.243;
   1:L PR[91] 10mm/sec CNT100;
   1:  PR[GP1:91,1] = PR[GP1:90,1] + -6.580;
   1:  PR[GP1:91,2] = PR[GP1:90,2] + -7.256;
   1:L PR[91] 10mm/sec CNT100;
   1:  PR[GP1:91,1] = PR[GP1:90,1] + -5.830;
   1:  PR[GP1:91,2] = PR[GP1:90,2] + -2.357;
   1:L PR[91] 10mm/sec CNT100;
   1:  PR[GP1:91,1] = PR[GP1:90,1] + -6.071;
   1:  PR[GP1:91,2] = PR[GP1:90,2] + -1.509;
   1:L PR[91] 10mm/sec CNT100;
   1:  PR[GP1:91,1] = PR[GP1:90,1] + 5.275;
   1:L PR[91] 10mm/sec CNT100;
   1:  PR[GP1:91,1] = PR[GP1:90,1] + 5.933;
   1:  PR[GP1:91,2] = PR[GP1:90,2] + -6.886;
   1:  PR[GP1:91,3] = PR[GP1:90,3] + 11.285;
   1:L PR[91] 10mm/sec CNT100;
   1:  PR[GP1:91,1] = PR[GP1:90,1] + 7.543;
   1:  PR[GP1:91,2] = PR[GP1:90,2] + -10.997;
   1:L PR[91] 10mm/sec CNT100;
   1:  PR[GP1:91,1] = PR[GP1:90,1] + 9.294;
   1:  PR[GP1:91,2] = PR[GP1:90,2] + -16.133;
   1:L PR[91] 10mm/sec CNT100;
   1:  PR[GP1:91,1] = PR[GP1:90,1] + 11.806;
   1:  PR[GP1:91,2] = PR[GP1:90,2] + -19.846;
   1:L PR[91] 10mm/sec CNT100;
   1:  PR[GP1:91,1] = PR[GP1:90,1] + 15.075;
   1:  PR[GP1:91,2] = PR[GP1:90,2] + -23.724;
   1:L PR[91] 10mm/sec CNT100;
   1:  PR[GP1:91,1] = PR[GP1:90,1] + 18.515;
   1:  PR[GP1:91,2] = PR[GP1:90,2] + -26.958;
   1:L PR[91] 10mm/sec CNT100;
   1:  PR[GP1:91,1] = PR[GP1:90,1] + 22.601;
   1:  PR[GP1:91,2] = PR[GP1:90,2] + -29.368;
   1:L PR[91] 10mm/sec CNT100;
   1:  PR[GP1:91,1] = PR[GP1:90,1] + 26.771;
   1:  PR[GP1:91,2] = PR[GP1:90,2] + -31.618;
   1:L PR[91] 10mm/sec CNT100;
   1:  PR[GP1:91,1] = PR[GP1:90,1] + 31.494;
   1:  PR[GP1:91,2] = PR[GP1:90,2] + -33.139;
   1:L PR[91] 10mm/sec CNT100;
   1:  PR[GP1:91,1] = PR[GP1:90,1] + 36.500;
   1:  PR[GP1:91,2] = PR[GP1:90,2] + -33.591;
   1:L PR[91] 10mm/sec CNT100;
   1:  PR[GP1:91,1] = PR[GP1:90,1] + 40.847;
   1:  PR[GP1:91,2] = PR[GP1:90,2] + -34.110;
   1:L PR[91] 10mm/sec CNT100;
   1:  PR[GP1:91,1] = PR[GP1:90,1] + 46.019;
   1:  PR[GP1:91,2] = PR[GP1:90,2] + -33.426;
   1:L PR[91] 10mm/sec CNT100;
   1:  PR[GP1:91,1] = PR[GP1:90,1] + 49.731;
   1:  PR[GP1:91,2] = PR[GP1:90,2] + -32.464;
   1:L PR[91] 10mm/sec CNT100;
   1:  PR[GP1:91,1] = PR[GP1:90,1] + 54.826;
   1:  PR[GP1:91,2] = PR[GP1:90,2] + -30.588;
   1:L PR[91] 10mm/sec CNT100;
   1:  PR[GP1:91,1] = PR[GP1:90,1] + 59.396;
   1:  PR[GP1:91,2] = PR[GP1:90,2] + -27.631;
   1:L PR[91] 10mm/sec CNT100;
   1:  PR[GP1:91,1] = PR[GP1:90,1] + 62.299;
   1:  PR[GP1:91,2] = PR[GP1:90,2] + -25.519;
   1:L PR[91] 10mm/sec CNT100;
   1:  PR[GP1:91,1] = PR[GP1:90,1] + 66.183;
   1:  PR[GP1:91,2] = PR[GP1:90,2] + -21.553;
   1:L PR[91] 10mm/sec CNT100;
   1:  PR[GP1:91,1] = PR[GP1:90,1] + 69.130;
   1:  PR[GP1:91,2] = PR[GP1:90,2] + -16.786;
   1:L PR[91] 10mm/sec CNT100;
   1:  PR[GP1:91,1] = PR[GP1:90,1] + 70.953;
   1:  PR[GP1:91,2] = PR[GP1:90,2] + -13.907;
   1:L PR[91] 10mm/sec CNT100;
   1:  PR[GP1:91,1] = PR[GP1:90,1] + 72.784;
   1:  PR[GP1:91,2] = PR[GP1:90,2] + -8.600;
   1:L PR[91] 10mm/sec CNT100;
   1:  PR[GP1:91,1] = PR[GP1:90,1] + 73.415;
   1:  PR[GP1:91,2] = PR[GP1:90,2] + -2.927;
   1:L PR[91] 10mm/sec CNT100;
   1:  PR[GP1:91,1] = PR[GP1:90,1] + 74.026;
   1:  PR[GP1:91,2] = PR[GP1:90,2] + 0.302;
   1:L PR[91] 10mm/sec CNT100;
   1:  PR[GP1:91,1] = PR[GP1:90,1] + 73.395;
   1:  PR[GP1:91,2] = PR[GP1:90,2] + 5.982;
   1:L PR[91] 10mm/sec CNT100;
   1:  PR[GP1:91,1] = PR[GP1:90,1] + 72.792;
   1:  PR[GP1:91,2] = PR[GP1:90,2] + 9.135;
   1:L PR[91] 10mm/sec CNT100;
   1:  PR[GP1:91,1] = PR[GP1:90,1] + 70.952;
   1:  PR[GP1:91,2] = PR[GP1:90,2] + 14.468;
   1:L PR[91] 10mm/sec CNT100;
   1:  PR[GP1:91,1] = PR[GP1:90,1] + 67.965;
   1:  PR[GP1:91,2] = PR[GP1:90,2] + 19.301;
   1:L PR[91] 10mm/sec CNT100;
   1:  PR[GP1:91,1] = PR[GP1:90,1] + 66.185;
   1:  PR[GP1:91,2] = PR[GP1:90,2] + 22.109;
   1:L PR[91] 10mm/sec CNT100;
   1:  PR[GP1:91,1] = PR[GP1:90,1] + 62.310;
   1:  PR[GP1:91,2] = PR[GP1:90,2] + 26.065;
   1:L PR[91] 10mm/sec CNT100;
   1:  PR[GP1:91,1] = PR[GP1:90,1] + 57.593;
   1:  PR[GP1:91,2] = PR[GP1:90,2] + 29.116;
   1:L PR[91] 10mm/sec CNT100;
   1:  PR[GP1:91,1] = PR[GP1:90,1] + 54.810;
   1:  PR[GP1:91,2] = PR[GP1:90,2] + 31.152;
   1:L PR[91] 10mm/sec CNT100;
   1:  PR[GP1:91,1] = PR[GP1:90,1] + 49.731;
   1:  PR[GP1:91,2] = PR[GP1:90,2] + 33.022;
   1:L PR[91] 10mm/sec CNT100;
   1:  PR[GP1:91,1] = PR[GP1:90,1] + 46.019;
   1:  PR[GP1:91,2] = PR[GP1:90,2] + 33.984;
   1:L PR[91] 10mm/sec CNT100;
   1:  PR[GP1:91,1] = PR[GP1:90,1] + 40.839;
   1:  PR[GP1:91,2] = PR[GP1:90,2] + 34.669;
   1:L PR[91] 10mm/sec CNT100;
   1:  PR[GP1:91,1] = PR[GP1:90,1] + 35.607;
   1:  PR[GP1:91,2] = PR[GP1:90,2] + 34.196;
   1:L PR[91] 10mm/sec CNT100;
   1:  PR[GP1:91,1] = PR[GP1:90,1] + 31.503;
   1:  PR[GP1:91,2] = PR[GP1:90,2] + 33.700;
   1:L PR[91] 10mm/sec CNT100;
   1:  PR[GP1:91,1] = PR[GP1:90,1] + 26.782;
   1:  PR[GP1:91,2] = PR[GP1:90,2] + 32.179;
   1:L PR[91] 10mm/sec CNT100;
   1:  PR[GP1:91,1] = PR[GP1:90,1] + 22.450;
   1:  PR[GP1:91,2] = PR[GP1:90,2] + 29.623;
   1:L PR[91] 10mm/sec CNT100;
   1:  PR[GP1:91,1] = PR[GP1:90,1] + 18.506;
   1:  PR[GP1:91,2] = PR[GP1:90,2] + 27.507;
   1:L PR[91] 10mm/sec CNT100;
   1:  PR[GP1:91,1] = PR[GP1:90,1] + 15.075;
   1:  PR[GP1:91,2] = PR[GP1:90,2] + 24.282;
   1:L PR[91] 10mm/sec CNT100;
   1:  PR[GP1:91,1] = PR[GP1:90,1] + 11.806;
   1:  PR[GP1:91,2] = PR[GP1:90,2] + 20.404;
   1:L PR[91] 10mm/sec CNT100;
   1:  PR[GP1:91,1] = PR[GP1:90,1] + 9.286;
   1:  PR[GP1:91,2] = PR[GP1:90,2] + 16.680;
   1:L PR[91] 10mm/sec CNT100;
   1:  PR[GP1:91,1] = PR[GP1:90,1] + 7.639;
   1:  PR[GP1:91,2] = PR[GP1:90,2] + 12.477;
   1:L PR[91] 10mm/sec CNT100;
   1:  PR[GP1:91,1] = PR[GP1:90,1] + 5.933;
   1:  PR[GP1:91,2] = PR[GP1:90,2] + 7.451;
   1:L PR[91] 10mm/sec CNT100;
   1:  PR[GP1:91,1] = PR[GP1:90,1] + 5.284;
   1:  PR[GP1:91,2] = PR[GP1:90,2] + 3.213;
   1:L PR[91] 10mm/sec CNT100;
   1:  PR[GP1:91,1] = PR[GP1:90,1] + 5.518;
   1:  PR[GP1:91,2] = PR[GP1:90,2] + 2.392;
   1:L PR[91] 10mm/sec CNT100;
   1:  PR[GP1:91,1] = PR[GP1:90,1] + -5.774;
   1:L PR[91] 10mm/sec CNT100;
   1:  PR[GP1:91,1] = PR[GP1:90,1] + -6.459;
   1:  PR[GP1:91,2] = PR[GP1:90,2] + 7.444;
   1:L PR[91] 10mm/sec CNT100;
   1:  PR[GP1:91,1] = PR[GP1:90,1] + -8.070;
   1:  PR[GP1:91,2] = PR[GP1:90,2] + 11.554;
   1:L PR[91] 10mm/sec CNT100;
   1:  PR[GP1:91,1] = PR[GP1:90,1] + -9.822;
   1:  PR[GP1:91,2] = PR[GP1:90,2] + 16.695;
   1:L PR[91] 10mm/sec CNT100;
   1:  PR[GP1:91,1] = PR[GP1:90,1] + -12.334;
   1:  PR[GP1:91,2] = PR[GP1:90,2] + 20.407;
   1:L PR[91] 10mm/sec CNT100;
   1:  PR[GP1:91,1] = PR[GP1:90,1] + -15.603;
   1:  PR[GP1:91,2] = PR[GP1:90,2] + 24.283;
   1:L PR[91] 10mm/sec CNT100;
   1:  PR[GP1:91,1] = PR[GP1:90,1] + -19.043;
   1:  PR[GP1:91,2] = PR[GP1:90,2] + 27.517;
   1:L PR[91] 10mm/sec CNT100;
   1:  PR[GP1:91,1] = PR[GP1:90,1] + -23.129;
   1:  PR[GP1:91,2] = PR[GP1:90,2] + 29.928;
   1:L PR[91] 10mm/sec CNT100;
   1:  PR[GP1:91,1] = PR[GP1:90,1] + -27.299;
   1:  PR[GP1:91,2] = PR[GP1:90,2] + 32.176;
   1:L PR[91] 10mm/sec CNT100;
   1:  PR[GP1:91,1] = PR[GP1:90,1] + -32.023;
   1:  PR[GP1:91,2] = PR[GP1:90,2] + 33.698;
   1:L PR[91] 10mm/sec CNT100;
   1:  PR[GP1:91,1] = PR[GP1:90,1] + -37.029;
   1:  PR[GP1:91,2] = PR[GP1:90,2] + 34.150;
   1:L PR[91] 10mm/sec CNT100;
   1:  PR[GP1:91,1] = PR[GP1:90,1] + -41.375;
   1:  PR[GP1:91,2] = PR[GP1:90,2] + 34.667;
   1:L PR[91] 10mm/sec CNT100;
   1:  PR[GP1:91,1] = PR[GP1:90,1] + -46.547;
   1:  PR[GP1:91,2] = PR[GP1:90,2] + 33.984;
   1:L PR[91] 10mm/sec CNT100;
   1:  PR[GP1:91,1] = PR[GP1:90,1] + -50.258;
   1:  PR[GP1:91,2] = PR[GP1:90,2] + 33.022;
   1:L PR[91] 10mm/sec CNT100;
   1:  PR[GP1:91,1] = PR[GP1:90,1] + -55.353;
   1:  PR[GP1:91,2] = PR[GP1:90,2] + 31.145;
   1:L PR[91] 10mm/sec CNT100;
   1:  PR[GP1:91,1] = PR[GP1:90,1] + -59.923;
   1:  PR[GP1:91,2] = PR[GP1:90,2] + 28.189;
   1:L PR[91] 10mm/sec CNT100;
   1:  PR[GP1:91,1] = PR[GP1:90,1] + -62.825;
   1:  PR[GP1:91,2] = PR[GP1:90,2] + 26.076;
   1:L PR[91] 10mm/sec CNT100;
   1:  PR[GP1:91,1] = PR[GP1:90,1] + -66.710;
   1:  PR[GP1:91,2] = PR[GP1:90,2] + 22.111;
   1:L PR[91] 10mm/sec CNT100;
   1:  PR[GP1:91,1] = PR[GP1:90,1] + -69.656;
   1:  PR[GP1:91,2] = PR[GP1:90,2] + 17.344;
   1:L PR[91] 10mm/sec CNT100;
   1:  PR[GP1:91,1] = PR[GP1:90,1] + -71.479;
   1:  PR[GP1:91,2] = PR[GP1:90,2] + 14.464;
   1:L PR[91] 10mm/sec CNT100;
   1:  PR[GP1:91,1] = PR[GP1:90,1] + -73.310;
   1:  PR[GP1:91,2] = PR[GP1:90,2] + 9.157;
   1:L PR[91] 10mm/sec CNT100;
   1:  PR[GP1:91,1] = PR[GP1:90,1] + -73.941;
   1:  PR[GP1:91,2] = PR[GP1:90,2] + 3.484;
   1:L PR[91] 10mm/sec CNT100;
   1:  PR[GP1:91,1] = PR[GP1:90,1] + -74.553;
   1:  PR[GP1:91,2] = PR[GP1:90,2] + 0.256;
   1:L PR[91] 10mm/sec CNT100;
   1:  PR[GP1:91,1] = PR[GP1:90,1] + -73.921;
   1:  PR[GP1:91,2] = PR[GP1:90,2] + -5.424;
   1:L PR[91] 10mm/sec CNT100;
   1:  PR[GP1:91,1] = PR[GP1:90,1] + -73.318;
   1:  PR[GP1:91,2] = PR[GP1:90,2] + -8.576;
   1:L PR[91] 10mm/sec CNT100;
   1:  PR[GP1:91,1] = PR[GP1:90,1] + -71.478;
   1:  PR[GP1:91,2] = PR[GP1:90,2] + -13.909;
   1:L PR[91] 10mm/sec CNT100;
   1:  PR[GP1:91,1] = PR[GP1:90,1] + -68.491;
   1:  PR[GP1:91,2] = PR[GP1:90,2] + -18.742;
   1:L PR[91] 10mm/sec CNT100;
   1:  PR[GP1:91,1] = PR[GP1:90,1] + -66.712;
   1:  PR[GP1:91,2] = PR[GP1:90,2] + -21.551;
   1:L PR[91] 10mm/sec CNT100;
   1:  PR[GP1:91,1] = PR[GP1:90,1] + -62.837;
   1:  PR[GP1:91,2] = PR[GP1:90,2] + -25.506;
   1:L PR[91] 10mm/sec CNT100;
   1:  PR[GP1:91,1] = PR[GP1:90,1] + -58.120;
   1:  PR[GP1:91,2] = PR[GP1:90,2] + -28.558;
   1:L PR[91] 10mm/sec CNT100;
   1:  PR[GP1:91,1] = PR[GP1:90,1] + -55.337;
   1:  PR[GP1:91,2] = PR[GP1:90,2] + -30.593;
   1:L PR[91] 10mm/sec CNT100;
   1:  PR[GP1:91,1] = PR[GP1:90,1] + -50.258;
   1:  PR[GP1:91,2] = PR[GP1:90,2] + -32.464;
   1:L PR[91] 10mm/sec CNT100;
   1:  PR[GP1:91,1] = PR[GP1:90,1] + -46.547;
   1:  PR[GP1:91,2] = PR[GP1:90,2] + -33.426;
   1:L PR[91] 10mm/sec CNT100;
   1:  PR[GP1:91,1] = PR[GP1:90,1] + -41.366;
   1:  PR[GP1:91,2] = PR[GP1:90,2] + -34.111;
   1:L PR[91] 10mm/sec CNT100;
   1:  PR[GP1:91,1] = PR[GP1:90,1] + -36.135;
   1:  PR[GP1:91,2] = PR[GP1:90,2] + -33.638;
   1:L PR[91] 10mm/sec CNT100;
   1:  PR[GP1:91,1] = PR[GP1:90,1] + -32.031;
   1:  PR[GP1:91,2] = PR[GP1:90,2] + -33.143;
   1:L PR[91] 10mm/sec CNT100;
   1:  PR[GP1:91,1] = PR[GP1:90,1] + -27.310;
   1:  PR[GP1:91,2] = PR[GP1:90,2] + -31.622;
   1:L PR[91] 10mm/sec CNT100;
   1:  PR[GP1:91,1] = PR[GP1:90,1] + -22.978;
   1:  PR[GP1:91,2] = PR[GP1:90,2] + -29.066;
   1:L PR[91] 10mm/sec CNT100;
   1:  PR[GP1:91,1] = PR[GP1:90,1] + -19.034;
   1:  PR[GP1:91,2] = PR[GP1:90,2] + -26.950;
   1:L PR[91] 10mm/sec CNT100;
   1:  PR[GP1:91,1] = PR[GP1:90,1] + -15.603;
   1:  PR[GP1:91,2] = PR[GP1:90,2] + -23.725;
   1:L PR[91] 10mm/sec CNT100;
   1:  PR[GP1:91,1] = PR[GP1:90,1] + -12.333;
   1:  PR[GP1:91,2] = PR[GP1:90,2] + -19.849;
   1:L PR[91] 10mm/sec CNT100;
   1:  PR[GP1:91,1] = PR[GP1:90,1] + -9.814;
   1:  PR[GP1:91,2] = PR[GP1:90,2] + -16.126;
   1:L PR[91] 10mm/sec CNT100;
   1:  PR[GP1:91,1] = PR[GP1:90,1] + -8.167;
   1:  PR[GP1:91,2] = PR[GP1:90,2] + -11.922;
   1:L PR[91] 10mm/sec CNT100;
   1:  PR[GP1:91,1] = PR[GP1:90,1] + -6.459;
   1:  PR[GP1:91,2] = PR[GP1:90,2] + -6.893;
   1:L PR[91] 10mm/sec CNT100;
   1:  PR[GP1:91,1] = PR[GP1:90,1] + -5.811;
   1:  PR[GP1:91,2] = PR[GP1:90,2] + -2.655;
   1:L PR[91] 10mm/sec CNT100;
   1:  PR[GP1:91,1] = PR[GP1:90,1] + -6.044;
   1:  PR[GP1:91,2] = PR[GP1:90,2] + -1.834;
   1:L PR[91] 10mm/sec CNT100;
   1:  PR[GP1:91,1] = PR[GP1:90,1] + 5.247;
   1:L PR[91] 10mm/sec CNT100;
   1:  PR[GP1:91,1] = PR[GP1:90,1] + 5.812;
   1:  PR[GP1:91,2] = PR[GP1:90,2] + -6.524;
   1:  PR[GP1:91,3] = PR[GP1:90,3] + 11.895;
   1:L PR[91] 10mm/sec CNT100;
   1:  PR[GP1:91,1] = PR[GP1:90,1] + 7.179;
   1:  PR[GP1:91,2] = PR[GP1:90,2] + -10.012;
   1:L PR[91] 10mm/sec CNT100;
   1:  PR[GP1:91,1] = PR[GP1:90,1] + 9.292;
   1:  PR[GP1:91,2] = PR[GP1:90,2] + -16.213;
   1:L PR[91] 10mm/sec CNT100;
   1:  PR[GP1:91,1] = PR[GP1:90,1] + 11.444;
   1:  PR[GP1:91,2] = PR[GP1:90,2] + -19.394;
   1:L PR[91] 10mm/sec CNT100;
   1:  PR[GP1:91,1] = PR[GP1:90,1] + 15.391;
   1:  PR[GP1:91,2] = PR[GP1:90,2] + -24.076;
   1:L PR[91] 10mm/sec CNT100;
   1:  PR[GP1:91,1] = PR[GP1:90,1] + 18.397;
   1:  PR[GP1:91,2] = PR[GP1:90,2] + -26.901;
   1:L PR[91] 10mm/sec CNT100;
   1:  PR[GP1:91,1] = PR[GP1:90,1] + 21.969;
   1:  PR[GP1:91,2] = PR[GP1:90,2] + -29.009;
   1:L PR[91] 10mm/sec CNT100;
   1:  PR[GP1:91,1] = PR[GP1:90,1] + 27.005;
   1:  PR[GP1:91,2] = PR[GP1:90,2] + -31.725;
   1:L PR[91] 10mm/sec CNT100;
   1:  PR[GP1:91,1] = PR[GP1:90,1] + 31.212;
   1:  PR[GP1:91,2] = PR[GP1:90,2] + -33.080;
   1:L PR[91] 10mm/sec CNT100;
   1:  PR[GP1:91,1] = PR[GP1:90,1] + 35.678;
   1:  PR[GP1:91,2] = PR[GP1:90,2] + -33.484;
   1:L PR[91] 10mm/sec CNT100;
   1:  PR[GP1:91,1] = PR[GP1:90,1] + 40.928;
   1:  PR[GP1:91,2] = PR[GP1:90,2] + -34.110;
   1:L PR[91] 10mm/sec CNT100;
   1:  PR[GP1:91,1] = PR[GP1:90,1] + 45.611;
   1:  PR[GP1:91,2] = PR[GP1:90,2] + -33.491;
   1:L PR[91] 10mm/sec CNT100;
   1:  PR[GP1:91,1] = PR[GP1:90,1] + 50.096;
   1:  PR[GP1:91,2] = PR[GP1:90,2] + -32.328;
   1:L PR[91] 10mm/sec CNT100;
   1:  PR[GP1:91,1] = PR[GP1:90,1] + 54.767;
   1:  PR[GP1:91,2] = PR[GP1:90,2] + -30.608;
   1:L PR[91] 10mm/sec CNT100;
   1:  PR[GP1:91,1] = PR[GP1:90,1] + 58.958;
   1:  PR[GP1:91,2] = PR[GP1:90,2] + -27.897;
   1:L PR[91] 10mm/sec CNT100;
   1:  PR[GP1:91,1] = PR[GP1:90,1] + 62.465;
   1:  PR[GP1:91,2] = PR[GP1:90,2] + -25.344;
   1:L PR[91] 10mm/sec CNT100;
   1:  PR[GP1:91,1] = PR[GP1:90,1] + 66.053;
   1:  PR[GP1:91,2] = PR[GP1:90,2] + -21.681;
   1:L PR[91] 10mm/sec CNT100;
   1:  PR[GP1:91,1] = PR[GP1:90,1] + 68.777;
   1:  PR[GP1:91,2] = PR[GP1:90,2] + -17.274;
   1:L PR[91] 10mm/sec CNT100;
   1:  PR[GP1:91,1] = PR[GP1:90,1] + 70.981;
   1:  PR[GP1:91,2] = PR[GP1:90,2] + -13.794;
   1:L PR[91] 10mm/sec CNT100;
   1:  PR[GP1:91,1] = PR[GP1:90,1] + 72.680;
   1:  PR[GP1:91,2] = PR[GP1:90,2] + -8.870;
   1:L PR[91] 10mm/sec CNT100;
   1:  PR[GP1:91,1] = PR[GP1:90,1] + 73.266;
   1:  PR[GP1:91,2] = PR[GP1:90,2] + -3.601;
   1:L PR[91] 10mm/sec CNT100;
   1:  PR[GP1:91,1] = PR[GP1:90,1] + 74.005;
